LIN {X 0,Y 489.55,Z 664.789,A -85,B 0,C 180,E1 -6475.471,E2 -6475.471} C_VEL
LIN {X 0,Y 489.917,Z 653.885,A -85,B 0,C 180,E1 -6476.402,E2 -6476.402} C_VEL
LIN {X 0,Y 490.26,Z 643.208,A -85,B 0,C 180,E1 -6477.124,E2 -6477.124} C_VEL
LIN {X 0,Y 490.656,Z 630.33,A -85,B 0,C 180,E1 -6477.794,E2 -6477.794} C_VEL
LIN {X 0,Y 490.871,Z 617.995,A -85,B 0,C 180,E1 -6478.256,E2 -6478.256} C_VEL
LIN {X 0,Y 491.024,Z 605.317,A -85,B 0,C 180,E1 -6478.565,E2 -6478.565} C_VEL
LIN {X 0,Y 491.793,Z 513.634,A -85,B 0,C 180,E1 -6480,E2 -6480} C_VEL
LIN {X 0,Y 489.493,Z 503.257,A -85,B 0,C 180,E1 -6480.257,E2 -6480.257} C_VEL
LIN {X 0,Y 488.87,Z 498.779,A -85,B 0,C 180,E1 -6481.39,E2 -6481.39} C_VEL
LIN {X 0,Y 488.953,Z 498.58,A -85,B 0,C 180,E1 -6482.471,E2 -6482.471} C_VEL
LIN {X 0,Y 488.865,Z 498.591,A -85,B 0,C 180,E1 -6485.775,E2 -6485.775} C_VEL
LIN {X 0,Y 488.809,Z 498.595,A -85,B 0,C 180,E1 -6488.266,E2 -6488.266} C_VEL
LIN {X 0,Y 488.823,Z 498.596,A -85,B 0,C 180,E1 -6491.612,E2 -6491.612} C_VEL
LIN {X 0,Y 488.752,Z 498.606,A -85,B 0,C 180,E1 -6495.001,E2 -6495.001} C_VEL
LIN {X 0,Y 488.745,Z 498.601,A -85,B 0,C 180,E1 -6498.442,E2 -6498.442} C_VEL
LIN {X 0,Y 488.698,Z 498.614,A -85,B 0,C 180,E1 -6501.071,E2 -6501.071} C_VEL
LIN {X 0,Y 488.685,Z 498.61,A -85,B 0,C 180,E1 -6503.746,E2 -6503.746} C_VEL
LIN {X 0,Y 488.791,Z 498.6,A -85,B 0,C 180,E1 -6506.946,E2 -6506.946} C_VEL
LIN {X 0,Y 488.711,Z 498.603,A -85,B 0,C 180,E1 -6510.365,E2 -6510.365} C_VEL
LIN {X 0,Y 488.729,Z 498.604,A -85,B 0,C 180,E1 -6513.485,E2 -6513.485} C_VEL
LIN {X 0,Y 488.683,Z 498.607,A -85,B 0,C 180,E1 -6516.356,E2 -6516.356} C_VEL
LIN {X 0,Y 488.696,Z 498.612,A -85,B 0,C 180,E1 -6519.255,E2 -6519.255} C_VEL
LIN {X 0,Y 488.703,Z 498.607,A -85,B 0,C 180,E1 -6521.601,E2 -6521.601} C_VEL
LIN {X 0,Y 488.707,Z 498.612,A -85,B 0,C 180,E1 -6524.802,E2 -6524.802} C_VEL
LIN {X 0,Y 488.691,Z 498.612,A -85,B 0,C 180,E1 -6527.476,E2 -6527.476} C_VEL
LIN {X 0,Y 488.729,Z 498.605,A -85,B 0,C 180,E1 -6529.677,E2 -6529.677} C_VEL
LIN {X 0,Y 488.679,Z 498.616,A -85,B 0,C 180,E1 -6532.842,E2 -6532.842} C_VEL
LIN {X 0,Y 488.732,Z 498.605,A -85,B 0,C 180,E1 -6535.888,E2 -6535.888} C_VEL
LIN {X 0,Y 488.693,Z 498.618,A -85,B 0,C 180,E1 -6538.821,E2 -6538.821} C_VEL
LIN {X 0,Y 488.744,Z 498.606,A -85,B 0,C 180,E1 -6541.672,E2 -6541.672} C_VEL
LIN {X 0,Y 488.775,Z 498.713,A -85,B 0,C 180,E1 -6542.836,E2 -6542.836} C_VEL
LIN {X 0,Y 491.08,Z 510.544,A -85,B 0,C 180,E1 -6544.802,E2 -6544.802} C_VEL
LIN {X 0,Y 490.719,Z 523.768,A -85,B 0,C 180,E1 -6546.812,E2 -6546.812} C_VEL
LIN {X 0,Y 490.136,Z 541.34,A -85,B 0,C 180,E1 -6549.434,E2 -6549.434} C_VEL
LIN {X 0,Y 489.49,Z 563.398,A -85,B 0,C 180,E1 -6552.667,E2 -6552.667} C_VEL
LIN {X 0,Y 489.298,Z 570.739,A -85,B 0,C 180,E1 -6553.729,E2 -6553.729} C_VEL
LIN {X 0,Y 491.608,Z 589.498,A -85,B 0,C 180,E1 -6554.105,E2 -6554.105} C_VEL
LIN {X 0,Y 490.867,Z 681.432,A -85,B 0,C 180,E1 -6555.543,E2 -6555.543} C_VEL
LIN {X 0,Y 490.515,Z 695.071,A -85,B 0,C 180,E1 -6555.929,E2 -6555.929} C_VEL
LIN {X 0,Y 490.122,Z 707.959,A -85,B 0,C 180,E1 -6556.473,E2 -6556.473} C_VEL
LIN {X 0,Y 489.729,Z 720.461,A -85,B 0,C 180,E1 -6557.19,E2 -6557.19} C_VEL
LIN {X 0,Y 489.426,Z 731.262,A -85,B 0,C 180,E1 -6557.983,E2 -6557.983} C_VEL
LIN {X 0,Y 489.029,Z 741.567,A -85,B 0,C 180,E1 -6558.918,E2 -6558.918} C_VEL
LIN {X 0,Y 488.714,Z 750.11,A -85,B 0,C 180,E1 -6559.854,E2 -6559.854} C_VEL
LIN {X 0,Y 488.44,Z 757.894,A -85,B 0,C 180,E1 -6560.893,E2 -6560.893} C_VEL
LIN {X 0,Y 488.234,Z 765.619,A -85,B 0,C 180,E1 -6562.14,E2 -6562.14} C_VEL
LIN {X 0,Y 488.086,Z 772.223,A -85,B 0,C 180,E1 -6563.485,E2 -6563.485} C_VEL
LIN {X 0,Y 488.065,Z 776.673,A -85,B 0,C 180,E1 -6564.629,E2 -6564.629} C_VEL
LIN {X 0,Y 488.014,Z 780.377,A -85,B 0,C 180,E1 -6565.871,E2 -6565.871} C_VEL
LIN {X 0,Y 487.975,Z 782.291,A -85,B 0,C 180,E1 -6566.697,E2 -6566.697} C_VEL
LIN {X 0,Y 487.988,Z 783.763,A -85,B 0,C 180,E1 -6567.524,E2 -6567.524} C_VEL
LIN {X 0,Y 487.892,Z 784.813,A -85,B 0,C 180,E1 -6568.349,E2 -6568.349} C_VEL
LIN {X 0,Y 487.843,Z 785.455,A -85,B 0,C 180,E1 -6569.175,E2 -6569.175} C_VEL
LIN {X 0,Y 487.839,Z 785.68,A -85,B 0,C 180,E1 -6570,E2 -6570} C_VEL
LIN {X 0,Y 487.842,Z 785.48,A -85,B 0,C 180,E1 -6570.825,E2 -6570.825} C_VEL
LIN {X 0,Y 487.892,Z 784.879,A -85,B 0,C 180,E1 -6571.651,E2 -6571.651} C_VEL
LIN {X 0,Y 487.988,Z 783.864,A -85,B 0,C 180,E1 -6572.476,E2 -6572.476} C_VEL
LIN {X 0,Y 487.972,Z 782.417,A -85,B 0,C 180,E1 -6573.303,E2 -6573.303} C_VEL
LIN {X 0,Y 487.944,Z 779.439,A -85,B 0,C 180,E1 -6574.544,E2 -6574.544} C_VEL
LIN {X 0,Y 488.087,Z 775.402,A -85,B 0,C 180,E1 -6575.785,E2 -6575.785} C_VEL
LIN {X 0,Y 488.182,Z 769.169,A -85,B 0,C 180,E1 -6577.236,E2 -6577.236} C_VEL
LIN {X 0,Y 488.359,Z 762.353,A -85,B 0,C 180,E1 -6578.482,E2 -6578.482} C_VEL
LIN {X 0,Y 488.599,Z 753.841,A -85,B 0,C 180,E1 -6579.73,E2 -6579.73} C_VEL
LIN {X 0,Y 488.895,Z 745.105,A -85,B 0,C 180,E1 -6580.77,E2 -6580.77} C_VEL
LIN {X 0,Y 489.313,Z 735.631,A -85,B 0,C 180,E1 -6581.705,E2 -6581.705} C_VEL
LIN {X 0,Y 489.655,Z 724.66,A -85,B 0,C 180,E1 -6582.577,E2 -6582.577} C_VEL
LIN {X 0,Y 490.05,Z 713.845,A -85,B 0,C 180,E1 -6583.265,E2 -6583.265} C_VEL
LIN {X 0,Y 490.399,Z 702.302,A -85,B 0,C 180,E1 -6583.836,E2 -6583.836} C_VEL
LIN {X 0,Y 490.741,Z 690.007,A -85,B 0,C 180,E1 -6584.276,E2 -6584.276} C_VEL
LIN {X 0,Y 490.992,Z 676.488,A -85,B 0,C 180,E1 -6584.586,E2 -6584.586} C_VEL
LIN {X 0,Y 491.55,Z 587.504,A -85,B 0,C 180,E1 -6585.947,E2 -6585.947} C_VEL
LIN {X 0,Y 489.411,Z 571.971,A -85,B 0,C 180,E1 -6586.265,E2 -6586.265} C_VEL
LIN {X 0,Y 490.118,Z 548.737,A -85,B 0,C 180,E1 -6589.692,E2 -6589.692} C_VEL
LIN {X 0,Y 490.772,Z 529.767,A -85,B 0,C 180,E1 -6592.523,E2 -6592.523} C_VEL
LIN {X 0,Y 491.452,Z 513.716,A -85,B 0,C 180,E1 -6594.952,E2 -6594.952} C_VEL
LIN {X 0,Y 491.047,Z 509.509,A -85,B 0,C 180,E1 -6595.621,E2 -6595.621} C_VEL
LIN {X 0,Y 488.771,Z 498.604,A -85,B 0,C 180,E1 -6597.452,E2 -6597.452} C_VEL
LIN {X 0,Y 488.709,Z 498.608,A -85,B 0,C 180,E1 -6600.362,E2 -6600.362} C_VEL
LIN {X 0,Y 488.733,Z 498.607,A -85,B 0,C 180,E1 -6603.483,E2 -6603.483} C_VEL
LIN {X 0,Y 488.679,Z 498.607,A -85,B 0,C 180,E1 -6606.354,E2 -6606.354} C_VEL
LIN {X 0,Y 488.698,Z 498.602,A -85,B 0,C 180,E1 -6609.253,E2 -6609.253} C_VEL
LIN {X 0,Y 488.72,Z 498.607,A -85,B 0,C 180,E1 -6611.601,E2 -6611.601} C_VEL
LIN {X 0,Y 488.707,Z 498.606,A -85,B 0,C 180,E1 -6614.801,E2 -6614.801} C_VEL
LIN {X 0,Y 488.686,Z 498.608,A -85,B 0,C 180,E1 -6617.474,E2 -6617.474} C_VEL
LIN {X 0,Y 488.727,Z 498.605,A -85,B 0,C 180,E1 -6619.676,E2 -6619.676} C_VEL
LIN {X 0,Y 488.673,Z 498.608,A -85,B 0,C 180,E1 -6622.277,E2 -6622.277} C_VEL
LIN {X 0,Y 488.722,Z 498.607,A -85,B 0,C 180,E1 -6625.051,E2 -6625.051} C_VEL
LIN {X 0,Y 488.699,Z 498.603,A -85,B 0,C 180,E1 -6628.045,E2 -6628.045} C_VEL
LIN {X 0,Y 488.726,Z 498.601,A -85,B 0,C 180,E1 -6630.73,E2 -6630.73} C_VEL
LIN {X 0,Y 488.758,Z 498.6,A -85,B 0,C 180,E1 -6633.528,E2 -6633.528} C_VEL
LIN {X 0,Y 488.684,Z 498.598,A -85,B 0,C 180,E1 -6636.254,E2 -6636.254} C_VEL
LIN {X 0,Y 488.737,Z 498.609,A -85,B 0,C 180,E1 -6639.175,E2 -6639.175} C_VEL
LIN {X 0,Y 488.75,Z 498.597,A -85,B 0,C 180,E1 -6641.627,E2 -6641.627} C_VEL
LIN {X 0,Y 488.752,Z 498.598,A -85,B 0,C 180,E1 -6644.999,E2 -6644.999} C_VEL
LIN {X 0,Y 488.822,Z 498.591,A -85,B 0,C 180,E1 -6648.388,E2 -6648.388} C_VEL
LIN {X 0,Y 488.809,Z 498.584,A -85,B 0,C 180,E1 -6651.734,E2 -6651.734} C_VEL
LIN {X 0,Y 488.863,Z 498.584,A -85,B 0,C 180,E1 -6654.225,E2 -6654.225} C_VEL
LIN {X 0,Y 488.952,Z 498.574,A -85,B 0,C 180,E1 -6657.529,E2 -6657.529} C_VEL
LIN {X 0,Y 488.959,Z 498.561,A -85,B 0,C 180,E1 -6660,E2 -6660} C_VEL
LIN {X 0,Y 488.953,Z 498.572,A -85,B 0,C 180,E1 -6662.472,E2 -6662.472} C_VEL
LIN {X 0,Y 488.864,Z 498.584,A -85,B 0,C 180,E1 -6665.776,E2 -6665.776} C_VEL
LIN {X 0,Y 488.809,Z 498.583,A -85,B 0,C 180,E1 -6668.267,E2 -6668.267} C_VEL
LIN {X 0,Y 488.799,Z 498.595,A -85,B 0,C 180,E1 -6671.613,E2 -6671.613} C_VEL
LIN {X 0,Y 488.753,Z 498.6,A -85,B 0,C 180,E1 -6675.001,E2 -6675.001} C_VEL
LIN {X 0,Y 488.747,Z 498.599,A -85,B 0,C 180,E1 -6678.443,E2 -6678.443} C_VEL
LIN {X 0,Y 488.7,Z 498.611,A -85,B 0,C 180,E1 -6681.071,E2 -6681.071} C_VEL
LIN {X 0,Y 488.686,Z 498.603,A -85,B 0,C 180,E1 -6683.746,E2 -6683.746} C_VEL
LIN {X 0,Y 488.792,Z 498.602,A -85,B 0,C 180,E1 -6686.946,E2 -6686.946} C_VEL
LIN {X 0,Y 488.713,Z 498.601,A -85,B 0,C 180,E1 -6690.366,E2 -6690.366} C_VEL
LIN {X 0,Y 488.731,Z 498.603,A -85,B 0,C 180,E1 -6693.485,E2 -6693.485} C_VEL
LIN {X 0,Y 488.686,Z 498.608,A -85,B 0,C 180,E1 -6696.357,E2 -6696.357} C_VEL
LIN {X 0,Y 488.698,Z 498.61,A -85,B 0,C 180,E1 -6699.255,E2 -6699.255} C_VEL
LIN {X 0,Y 488.705,Z 498.609,A -85,B 0,C 180,E1 -6701.601,E2 -6701.601} C_VEL
LIN {X 0,Y 488.699,Z 498.606,A -85,B 0,C 180,E1 -6704.025,E2 -6704.025} C_VEL
LIN {X 0,Y 488.731,Z 498.608,A -85,B 0,C 180,E1 -6707.172,E2 -6707.172} C_VEL
LIN {X 0,Y 488.731,Z 498.603,A -85,B 0,C 180,E1 -6709.678,E2 -6709.678} C_VEL
LIN {X 0,Y 488.679,Z 498.615,A -85,B 0,C 180,E1 -6712.842,E2 -6712.842} C_VEL
LIN {X 0,Y 488.731,Z 498.603,A -85,B 0,C 180,E1 -6715.888,E2 -6715.888} C_VEL
LIN {X 0,Y 488.693,Z 498.611,A -85,B 0,C 180,E1 -6718.821,E2 -6718.821} C_VEL
LIN {X 0,Y 488.746,Z 498.603,A -85,B 0,C 180,E1 -6721.672,E2 -6721.672} C_VEL
LIN {X 0,Y 488.796,Z 498.602,A -85,B 0,C 180,E1 -6723.111,E2 -6723.111} C_VEL
LIN {X 0,Y 488.575,Z 499.275,A -85,B 0,C 180,E1 -6723.566,E2 -6723.566} C_VEL
LIN {X 0,Y 487.813,Z 501.458,A -85,B 0,C 180,E1 -6724.088,E2 -6724.088} C_VEL
LIN {X 0,Y 483.782,Z 512.802,A -85,B 0,C 180,E1 -6725.858,E2 -6725.858} C_VEL
LIN {X 0,Y 483.468,Z 515.113,A -85,B 0,C 180,E1 -6726.244,E2 -6726.244} C_VEL
LIN {X 0,Y 482.892,Z 533.439,A -85,B 0,C 180,E1 -6729.334,E2 -6729.334} C_VEL
LIN {X 0,Y 482.591,Z 546.967,A -85,B 0,C 180,E1 -6731.548,E2 -6731.548} C_VEL
LIN {X 0,Y 484.969,Z 561.064,A -85,B 0,C 180,E1 -6731.847,E2 -6731.847} C_VEL
LIN {X 0,Y 484.263,Z 656.005,A -85,B 0,C 180,E1 -6733.283,E2 -6733.283} C_VEL
LIN {X 0,Y 484.057,Z 669.122,A -85,B 0,C 180,E1 -6733.65,E2 -6733.65} C_VEL
LIN {X 0,Y 483.687,Z 681.903,A -85,B 0,C 180,E1 -6734.191,E2 -6734.191} C_VEL
LIN {X 0,Y 483.287,Z 693.124,A -85,B 0,C 180,E1 -6734.826,E2 -6734.826} C_VEL
LIN {X 0,Y 482.888,Z 703.46,A -85,B 0,C 180,E1 -6735.568,E2 -6735.568} C_VEL
LIN {X 0,Y 482.393,Z 714.084,A -85,B 0,C 180,E1 -6736.52,E2 -6736.52} C_VEL
LIN {X 0,Y 481.997,Z 724.342,A -85,B 0,C 180,E1 -6737.671,E2 -6737.671} C_VEL
LIN {X 0,Y 481.688,Z 732.834,A -85,B 0,C 180,E1 -6738.854,E2 -6738.854} C_VEL
LIN {X 0,Y 481.31,Z 740.173,A -85,B 0,C 180,E1 -6740.121,E2 -6740.121} C_VEL
LIN {X 0,Y 481.096,Z 746.945,A -85,B 0,C 180,E1 -6741.6,E2 -6741.6} C_VEL
LIN {X 0,Y 480.994,Z 751.387,A -85,B 0,C 180,E1 -6742.866,E2 -6742.866} C_VEL
LIN {X 0,Y 480.926,Z 754.743,A -85,B 0,C 180,E1 -6744.129,E2 -6744.129} C_VEL
LIN {X 0,Y 480.791,Z 757.67,A -85,B 0,C 180,E1 -6745.809,E2 -6745.809} C_VEL
LIN {X 0,Y 480.871,Z 758.544,A -85,B 0,C 180,E1 -6746.649,E2 -6746.649} C_VEL
LIN {X 0,Y 480.821,Z 759.001,A -85,B 0,C 180,E1 -6747.487,E2 -6747.487} C_VEL
LIN {X 0,Y 480.822,Z 759.052,A -85,B 0,C 180,E1 -6748.325,E2 -6748.325} C_VEL
LIN {X 0,Y 480.746,Z 758.024,A -85,B 0,C 180,E1 -6750,E2 -6750} C_VEL
LIN {X 0,Y 480.766,Z 756.885,A -85,B 0,C 180,E1 -6750.838,E2 -6750.838} C_VEL
LIN {X 0,Y 480.852,Z 755.339,A -85,B 0,C 180,E1 -6751.675,E2 -6751.675} C_VEL
LIN {X 0,Y 481.015,Z 752.226,A -85,B 0,C 180,E1 -6752.931,E2 -6752.931} C_VEL
LIN {X 0,Y 481.122,Z 748.071,A -85,B 0,C 180,E1 -6754.188,E2 -6754.188} C_VEL
LIN {X 0,Y 481.265,Z 741.773,A -85,B 0,C 180,E1 -6755.657,E2 -6755.657} C_VEL
LIN {X 0,Y 481.628,Z 735.259,A -85,B 0,C 180,E1 -6756.847,E2 -6756.847} C_VEL
LIN {X 0,Y 481.836,Z 727.805,A -85,B 0,C 180,E1 -6757.965,E2 -6757.965} C_VEL
LIN {X 0,Y 482.203,Z 719.295,A -85,B 0,C 180,E1 -6759.014,E2 -6759.014} C_VEL
LIN {X 0,Y 482.734,Z 708.869,A -85,B 0,C 180,E1 -6760.061,E2 -6760.061} C_VEL
LIN {X 0,Y 483.098,Z 698.445,A -85,B 0,C 180,E1 -6760.901,E2 -6760.901} C_VEL
LIN {X 0,Y 483.527,Z 686.901,A -85,B 0,C 180,E1 -6761.634,E2 -6761.634} C_VEL
LIN {X 0,Y 483.921,Z 675.067,A -85,B 0,C 180,E1 -6762.209,E2 -6762.209} C_VEL
LIN {X 0,Y 484.148,Z 662.145,A -85,B 0,C 180,E1 -6762.656,E2 -6762.656} C_VEL
LIN {X 0,Y 484.376,Z 648.3,A -85,B 0,C 180,E1 -6762.943,E2 -6762.943} C_VEL
LIN {X 0,Y 484.876,Z 560.303,A -85,B 0,C 180,E1 -6764.254,E2 -6764.254} C_VEL
LIN {X 0,Y 482.563,Z 546.856,A -85,B 0,C 180,E1 -6764.55,E2 -6764.55} C_VEL
LIN {X 0,Y 482.963,Z 529.781,A -85,B 0,C 180,E1 -6767.356,E2 -6767.356} C_VEL
LIN {X 0,Y 483.545,Z 510.287,A -85,B 0,C 180,E1 -6770.637,E2 -6770.637} C_VEL
LIN {X 0,Y 482.503,Z 503.71,A -85,B 0,C 180,E1 -6771.803,E2 -6771.803} C_VEL
LIN {X 0,Y 481.685,Z 499.49,A -85,B 0,C 180,E1 -6772.576,E2 -6772.576} C_VEL
LIN {X 0,Y 481.703,Z 499.481,A -85,B 0,C 180,E1 -6775.956,E2 -6775.956} C_VEL
LIN {X 0,Y 481.702,Z 499.485,A -85,B 0,C 180,E1 -6778.781,E2 -6778.781} C_VEL
LIN {X 0,Y 481.66,Z 499.486,A -85,B 0,C 180,E1 -6782.189,E2 -6782.189} C_VEL
LIN {X 0,Y 481.689,Z 499.483,A -85,B 0,C 180,E1 -6784.681,E2 -6784.681} C_VEL
LIN {X 0,Y 481.655,Z 499.484,A -85,B 0,C 180,E1 -6788.006,E2 -6788.006} C_VEL
LIN {X 0,Y 481.661,Z 499.488,A -85,B 0,C 180,E1 -6791.04,E2 -6791.04} C_VEL
LIN {X 0,Y 481.68,Z 499.483,A -85,B 0,C 180,E1 -6793.294,E2 -6793.294} C_VEL
LIN {X 0,Y 481.68,Z 499.485,A -85,B 0,C 180,E1 -6796.845,E2 -6796.845} C_VEL
LIN {X 0,Y 481.673,Z 499.483,A -85,B 0,C 180,E1 -6800.059,E2 -6800.059} C_VEL
LIN {X 0,Y 481.626,Z 499.491,A -85,B 0,C 180,E1 -6803.253,E2 -6803.253} C_VEL
LIN {X 0,Y 481.704,Z 499.484,A -85,B 0,C 180,E1 -6806.329,E2 -6806.329} C_VEL
LIN {X 0,Y 481.74,Z 499.495,A -85,B 0,C 180,E1 -6806.957,E2 -6806.957} C_VEL
LIN {X 0,Y 482.178,Z 502.037,A -85,B 0,C 180,E1 -6807.573,E2 -6807.573} C_VEL
LIN {X 0,Y 484.86,Z 513.987,A -85,B 0,C 180,E1 -6807.872,E2 -6807.872} C_VEL
LIN {X 0,Y 484.13,Z 608.315,A -85,B 0,C 180,E1 -6809.374,E2 -6809.374} C_VEL
LIN {X 0,Y 483.883,Z 621.472,A -85,B 0,C 180,E1 -6809.747,E2 -6809.747} C_VEL
LIN {X 0,Y 483.679,Z 633.972,A -85,B 0,C 180,E1 -6810.274,E2 -6810.274} C_VEL
LIN {X 0,Y 483.265,Z 646.179,A -85,B 0,C 180,E1 -6810.971,E2 -6810.971} C_VEL
LIN {X 0,Y 482.841,Z 657.038,A -85,B 0,C 180,E1 -6811.767,E2 -6811.767} C_VEL
LIN {X 0,Y 482.479,Z 667.159,A -85,B 0,C 180,E1 -6812.689,E2 -6812.689} C_VEL
LIN {X 0,Y 482.039,Z 677.233,A -85,B 0,C 180,E1 -6813.83,E2 -6813.83} C_VEL
LIN {X 0,Y 481.745,Z 685.374,A -85,B 0,C 180,E1 -6814.971,E2 -6814.971} C_VEL
LIN {X 0,Y 481.441,Z 693.216,A -85,B 0,C 180,E1 -6816.331,E2 -6816.331} C_VEL
LIN {X 0,Y 481.224,Z 699.311,A -85,B 0,C 180,E1 -6817.684,E2 -6817.684} C_VEL
LIN {X 0,Y 481.072,Z 704.569,A -85,B 0,C 180,E1 -6819.221,E2 -6819.221} C_VEL
LIN {X 0,Y 480.916,Z 707.444,A -85,B 0,C 180,E1 -6820.359,E2 -6820.359} C_VEL
LIN {X 0,Y 480.871,Z 709.94,A -85,B 0,C 180,E1 -6821.798,E2 -6821.798} C_VEL
LIN {X 0,Y 480.793,Z 711.099,A -85,B 0,C 180,E1 -6823.001,E2 -6823.001} C_VEL
LIN {X 0,Y 480.822,Z 711.43,A -85,B 0,C 180,E1 -6823.876,E2 -6823.876} C_VEL
LIN {X 0,Y 480.845,Z 711.334,A -85,B 0,C 180,E1 -6824.746,E2 -6824.746} C_VEL
LIN {X 0,Y 480.851,Z 710.776,A -85,B 0,C 180,E1 -6825.613,E2 -6825.613} C_VEL
LIN {X 0,Y 480.875,Z 709.814,A -85,B 0,C 180,E1 -6826.476,E2 -6826.476} C_VEL
LIN {X 0,Y 480.953,Z 708.435,A -85,B 0,C 180,E1 -6827.338,E2 -6827.338} C_VEL
LIN {X 0,Y 481.043,Z 705.478,A -85,B 0,C 180,E1 -6828.634,E2 -6828.634} C_VEL
LIN {X 0,Y 481.174,Z 701.505,A -85,B 0,C 180,E1 -6829.905,E2 -6829.905} C_VEL
LIN {X 0,Y 481.426,Z 695.323,A -85,B 0,C 180,E1 -6831.394,E2 -6831.394} C_VEL
LIN {X 0,Y 481.726,Z 687.998,A -85,B 0,C 180,E1 -6832.766,E2 -6832.766} C_VEL
LIN {X 0,Y 482.039,Z 680.194,A -85,B 0,C 180,E1 -6833.932,E2 -6833.932} C_VEL
LIN {X 0,Y 482.302,Z 671.585,A -85,B 0,C 180,E1 -6834.984,E2 -6834.984} C_VEL
LIN {X 0,Y 482.745,Z 660.949,A -85,B 0,C 180,E1 -6836.034,E2 -6836.034} C_VEL
LIN {X 0,Y 483.169,Z 650.341,A -85,B 0,C 180,E1 -6836.873,E2 -6836.873} C_VEL
LIN {X 0,Y 483.496,Z 640.424,A -85,B 0,C 180,E1 -6837.5,E2 -6837.5} C_VEL
LIN {X 0,Y 483.794,Z 627.481,A -85,B 0,C 180,E1 -6838.127,E2 -6838.127} C_VEL
LIN {X 0,Y 484.089,Z 614.439,A -85,B 0,C 180,E1 -6838.57,E2 -6838.57} C_VEL
LIN {X 0,Y 484.219,Z 601.944,A -85,B 0,C 180,E1 -6838.83,E2 -6838.83} C_VEL
LIN {X 0,Y 484.924,Z 514.261,A -85,B 0,C 180,E1 -6840.233,E2 -6840.233} C_VEL
LIN {X 0,Y 482.552,Z 503.84,A -85,B 0,C 180,E1 -6840.524,E2 -6840.524} C_VEL
LIN {X 0,Y 481.804,Z 499.472,A -85,B 0,C 180,E1 -6841.672,E2 -6841.672} C_VEL
LIN {X 0,Y 481.92,Z 499.456,A -85,B 0,C 180,E1 -6842.507,E2 -6842.507} C_VEL
LIN {X 0,Y 481.823,Z 499.468,A -85,B 0,C 180,E1 -6845.86,E2 -6845.86} C_VEL
LIN {X 0,Y 481.755,Z 499.474,A -85,B 0,C 180,E1 -6848.388,E2 -6848.388} C_VEL
LIN {X 0,Y 481.786,Z 499.471,A -85,B 0,C 180,E1 -6851.784,E2 -6851.784} C_VEL
LIN {X 0,Y 481.733,Z 499.481,A -85,B 0,C 180,E1 -6855.224,E2 -6855.224} C_VEL
LIN {X 0,Y 481.703,Z 499.48,A -85,B 0,C 180,E1 -6858.722,E2 -6858.722} C_VEL
LIN {X 0,Y 481.638,Z 499.491,A -85,B 0,C 180,E1 -6861.395,E2 -6861.395} C_VEL
LIN {X 0,Y 481.668,Z 499.482,A -85,B 0,C 180,E1 -6864.114,E2 -6864.114} C_VEL
LIN {X 0,Y 481.744,Z 499.478,A -85,B 0,C 180,E1 -6867.141,E2 -6867.141} C_VEL
LIN {X 0,Y 481.681,Z 499.48,A -85,B 0,C 180,E1 -6869.741,E2 -6869.741} C_VEL
LIN {X 0,Y 481.666,Z 499.483,A -85,B 0,C 180,E1 -6872.675,E2 -6872.675} C_VEL
LIN {X 0,Y 481.636,Z 499.485,A -85,B 0,C 180,E1 -6875.71,E2 -6875.71} C_VEL
LIN {X 0,Y 481.686,Z 499.485,A -85,B 0,C 180,E1 -6878.858,E2 -6878.858} C_VEL
LIN {X 0,Y 481.642,Z 499.486,A -85,B 0,C 180,E1 -6882.161,E2 -6882.161} C_VEL
LIN {X 0,Y 481.655,Z 499.487,A -85,B 0,C 180,E1 -6885.544,E2 -6885.544} C_VEL
LIN {X 0,Y 481.658,Z 499.486,A -85,B 0,C 180,E1 -6888.087,E2 -6888.087} C_VEL
LIN {X 0,Y 481.668,Z 499.488,A -85,B 0,C 180,E1 -6891.142,E2 -6891.142} C_VEL
LIN {X 0,Y 481.664,Z 499.491,A -85,B 0,C 180,E1 -6894.796,E2 -6894.796} C_VEL
LIN {X 0,Y 481.671,Z 499.49,A -85,B 0,C 180,E1 -6897.327,E2 -6897.327} C_VEL
LIN {X 0,Y 481.678,Z 499.488,A -85,B 0,C 180,E1 -6900.26,E2 -6900.26} C_VEL
LIN {X 0,Y 481.724,Z 499.583,A -85,B 0,C 180,E1 -6902.602,E2 -6902.602} C_VEL
LIN {X 0,Y 484.129,Z 511.692,A -85,B 0,C 180,E1 -6904.663,E2 -6904.663} C_VEL
LIN {X 0,Y 483.869,Z 522.387,A -85,B 0,C 180,E1 -6906.326,E2 -6906.326} C_VEL
LIN {X 0,Y 483.155,Z 542.273,A -85,B 0,C 180,E1 -6909.345,E2 -6909.345} C_VEL
LIN {X 0,Y 482.459,Z 564.242,A -85,B 0,C 180,E1 -6912.625,E2 -6912.625} C_VEL
LIN {X 0,Y 482.318,Z 569.981,A -85,B 0,C 180,E1 -6913.474,E2 -6913.474} C_VEL
LIN {X 0,Y 484.758,Z 589.981,A -85,B 0,C 180,E1 -6913.892,E2 -6913.892} C_VEL
LIN {X 0,Y 483.996,Z 680.253,A -85,B 0,C 180,E1 -6915.333,E2 -6915.333} C_VEL
LIN {X 0,Y 483.622,Z 693.277,A -85,B 0,C 180,E1 -6915.698,E2 -6915.698} C_VEL
LIN {X 0,Y 483.236,Z 705.973,A -85,B 0,C 180,E1 -6916.223,E2 -6916.223} C_VEL
LIN {X 0,Y 482.806,Z 717.844,A -85,B 0,C 180,E1 -6916.886,E2 -6916.886} C_VEL
LIN {X 0,Y 482.494,Z 729.198,A -85,B 0,C 180,E1 -6917.687,E2 -6917.687} C_VEL
LIN {X 0,Y 482.054,Z 740.067,A -85,B 0,C 180,E1 -6918.649,E2 -6918.649} C_VEL
LIN {X 0,Y 481.677,Z 749.678,A -85,B 0,C 180,E1 -6919.704,E2 -6919.704} C_VEL
LIN {X 0,Y 481.387,Z 757.526,A -85,B 0,C 180,E1 -6920.759,E2 -6920.759} C_VEL
LIN {X 0,Y 481.174,Z 765.167,A -85,B 0,C 180,E1 -6922.024,E2 -6922.024} C_VEL
LIN {X 0,Y 481.017,Z 771.283,A -85,B 0,C 180,E1 -6923.288,E2 -6923.288} C_VEL
LIN {X 0,Y 481.001,Z 776.127,A -85,B 0,C 180,E1 -6924.55,E2 -6924.55} C_VEL
LIN {X 0,Y 480.911,Z 779.792,A -85,B 0,C 180,E1 -6925.81,E2 -6925.81} C_VEL
LIN {X 0,Y 480.903,Z 781.715,A -85,B 0,C 180,E1 -6926.649,E2 -6926.649} C_VEL
LIN {X 0,Y 480.925,Z 783.201,A -85,B 0,C 180,E1 -6927.487,E2 -6927.487} C_VEL
LIN {X 0,Y 480.825,Z 784.256,A -85,B 0,C 180,E1 -6928.325,E2 -6928.325} C_VEL
LIN {X 0,Y 480.769,Z 784.905,A -85,B 0,C 180,E1 -6929.162,E2 -6929.162} C_VEL
LIN {X 0,Y 480.761,Z 785.14,A -85,B 0,C 180,E1 -6930,E2 -6930} C_VEL
LIN {X 0,Y 480.768,Z 784.944,A -85,B 0,C 180,E1 -6930.838,E2 -6930.838} C_VEL
LIN {X 0,Y 480.825,Z 784.339,A -85,B 0,C 180,E1 -6931.675,E2 -6931.675} C_VEL
LIN {X 0,Y 480.925,Z 783.322,A -85,B 0,C 180,E1 -6932.513,E2 -6932.513} C_VEL
LIN {X 0,Y 480.899,Z 781.872,A -85,B 0,C 180,E1 -6933.351,E2 -6933.351} C_VEL
LIN {X 0,Y 480.859,Z 778.887,A -85,B 0,C 180,E1 -6934.611,E2 -6934.611} C_VEL
LIN {X 0,Y 480.983,Z 774.845,A -85,B 0,C 180,E1 -6935.87,E2 -6935.87} C_VEL
LIN {X 0,Y 481.107,Z 768.598,A -85,B 0,C 180,E1 -6937.343,E2 -6937.343} C_VEL
LIN {X 0,Y 481.292,Z 761.756,A -85,B 0,C 180,E1 -6938.608,E2 -6938.608} C_VEL
LIN {X 0,Y 481.534,Z 753.224,A -85,B 0,C 180,E1 -6939.874,E2 -6939.874} C_VEL
LIN {X 0,Y 481.871,Z 744.459,A -85,B 0,C 180,E1 -6940.929,E2 -6940.929} C_VEL
LIN {X 0,Y 482.235,Z 735.012,A -85,B 0,C 180,E1 -6941.875,E2 -6941.875} C_VEL
LIN {X 0,Y 482.72,Z 723.355,A -85,B 0,C 180,E1 -6942.806,E2 -6942.806} C_VEL
LIN {X 0,Y 483.146,Z 711.178,A -85,B 0,C 180,E1 -6943.565,E2 -6943.565} C_VEL
LIN {X 0,Y 483.502,Z 698.859,A -85,B 0,C 180,E1 -6944.145,E2 -6944.145} C_VEL
LIN {X 0,Y 483.952,Z 685.369,A -85,B 0,C 180,E1 -6944.588,E2 -6944.588} C_VEL
LIN {X 0,Y 484.139,Z 670.223,A -85,B 0,C 180,E1 -6944.878,E2 -6944.878} C_VEL
LIN {X 0,Y 484.74,Z 588.484,A -85,B 0,C 180,E1 -6946.153,E2 -6946.153} C_VEL
LIN {X 0,Y 482.417,Z 571.336,A -85,B 0,C 180,E1 -6946.531,E2 -6946.531} C_VEL
LIN {X 0,Y 483.182,Z 548.255,A -85,B 0,C 180,E1 -6949.987,E2 -6949.987} C_VEL
LIN {X 0,Y 483.902,Z 529.32,A -85,B 0,C 180,E1 -6952.861,E2 -6952.861} C_VEL
LIN {X 0,Y 484.532,Z 514.74,A -85,B 0,C 180,E1 -6955.103,E2 -6955.103} C_VEL
LIN {X 0,Y 483.697,Z 508.822,A -85,B 0,C 180,E1 -6956.073,E2 -6956.073} C_VEL
LIN {X 0,Y 481.744,Z 499.48,A -85,B 0,C 180,E1 -6957.699,E2 -6957.699} C_VEL
LIN {X 0,Y 481.645,Z 499.49,A -85,B 0,C 180,E1 -6960.71,E2 -6960.71} C_VEL
LIN {X 0,Y 481.695,Z 499.482,A -85,B 0,C 180,E1 -6963.732,E2 -6963.732} C_VEL
LIN {X 0,Y 481.623,Z 499.489,A -85,B 0,C 180,E1 -6966.746,E2 -6966.746} C_VEL
LIN {X 0,Y 481.673,Z 499.48,A -85,B 0,C 180,E1 -6969.94,E2 -6969.94} C_VEL
LIN {X 0,Y 481.676,Z 499.484,A -85,B 0,C 180,E1 -6973.294,E2 -6973.294} C_VEL
LIN {X 0,Y 481.634,Z 499.49,A -85,B 0,C 180,E1 -6976.7,E2 -6976.7} C_VEL
LIN {X 0,Y 481.681,Z 499.481,A -85,B 0,C 180,E1 -6980.06,E2 -6980.06} C_VEL
LIN {X 0,Y 481.623,Z 499.488,A -85,B 0,C 180,E1 -6983.253,E2 -6983.253} C_VEL
LIN {X 0,Y 481.702,Z 499.478,A -85,B 0,C 180,E1 -6986.329,E2 -6986.329} C_VEL
LIN {X 0,Y 481.651,Z 499.483,A -85,B 0,C 180,E1 -6989.415,E2 -6989.415} C_VEL
LIN {X 0,Y 481.695,Z 499.478,A -85,B 0,C 180,E1 -6992.168,E2 -6992.168} C_VEL
LIN {X 0,Y 481.71,Z 499.478,A -85,B 0,C 180,E1 -6994.97,E2 -6994.97} C_VEL
LIN {X 0,Y 481.641,Z 499.485,A -85,B 0,C 180,E1 -6997.704,E2 -6997.704} C_VEL
LIN {X 0,Y 481.699,Z 499.478,A -85,B 0,C 180,E1 -7000.393,E2 -7000.393} C_VEL
LIN {X 0,Y 481.682,Z 499.477,A -85,B 0,C 180,E1 -7003.034,E2 -7003.034} C_VEL
LIN {X 0,Y 481.68,Z 499.481,A -85,B 0,C 180,E1 -7005.639,E2 -7005.639} C_VEL
LIN {X 0,Y 481.786,Z 499.467,A -85,B 0,C 180,E1 -7008.216,E2 -7008.216} C_VEL
LIN {X 0,Y 481.754,Z 499.463,A -85,B 0,C 180,E1 -7011.612,E2 -7011.612} C_VEL
LIN {X 0,Y 481.822,Z 499.461,A -85,B 0,C 180,E1 -7014.14,E2 -7014.14} C_VEL
LIN {X 0,Y 481.919,Z 499.45,A -85,B 0,C 180,E1 -7017.493,E2 -7017.493} C_VEL
LIN {X 0,Y 481.93,Z 499.436,A -85,B 0,C 180,E1 -7020,E2 -7020} C_VEL
LIN {X 0,Y 481.92,Z 499.449,A -85,B 0,C 180,E1 -7022.508,E2 -7022.508} C_VEL
LIN {X 0,Y 481.823,Z 499.461,A -85,B 0,C 180,E1 -7025.861,E2 -7025.861} C_VEL
LIN {X 0,Y 481.755,Z 499.461,A -85,B 0,C 180,E1 -7028.389,E2 -7028.389} C_VEL
LIN {X 0,Y 481.744,Z 499.473,A -85,B 0,C 180,E1 -7031.785,E2 -7031.785} C_VEL
LIN {X 0,Y 481.733,Z 499.47,A -85,B 0,C 180,E1 -7035.225,E2 -7035.225} C_VEL
LIN {X 0,Y 481.704,Z 499.479,A -85,B 0,C 180,E1 -7038.722,E2 -7038.722} C_VEL
LIN {X 0,Y 481.639,Z 499.486,A -85,B 0,C 180,E1 -7041.395,E2 -7041.395} C_VEL
LIN {X 0,Y 481.67,Z 499.476,A -85,B 0,C 180,E1 -7044.114,E2 -7044.114} C_VEL
LIN {X 0,Y 481.745,Z 499.478,A -85,B 0,C 180,E1 -7047.141,E2 -7047.141} C_VEL
LIN {X 0,Y 481.682,Z 499.476,A -85,B 0,C 180,E1 -7049.741,E2 -7049.741} C_VEL
LIN {X 0,Y 481.668,Z 499.486,A -85,B 0,C 180,E1 -7052.675,E2 -7052.675} C_VEL
LIN {X 0,Y 481.639,Z 499.486,A -85,B 0,C 180,E1 -7055.71,E2 -7055.71} C_VEL
LIN {X 0,Y 481.668,Z 499.489,A -85,B 0,C 180,E1 -7058.86,E2 -7058.86} C_VEL
LIN {X 0,Y 481.651,Z 499.487,A -85,B 0,C 180,E1 -7061.914,E2 -7061.914} C_VEL
LIN {X 0,Y 481.657,Z 499.485,A -85,B 0,C 180,E1 -7064.458,E2 -7064.458} C_VEL
LIN {X 0,Y 481.682,Z 499.486,A -85,B 0,C 180,E1 -7066.847,E2 -7066.847} C_VEL
LIN {X 0,Y 481.676,Z 499.481,A -85,B 0,C 180,E1 -7070.061,E2 -7070.061} C_VEL
LIN {X 0,Y 481.625,Z 499.493,A -85,B 0,C 180,E1 -7073.254,E2 -7073.254} C_VEL
LIN {X 0,Y 481.71,Z 499.479,A -85,B 0,C 180,E1 -7076.331,E2 -7076.331} C_VEL
LIN {X 0,Y 481.652,Z 499.488,A -85,B 0,C 180,E1 -7079.418,E2 -7079.418} C_VEL
LIN {X 0,Y 481.702,Z 499.48,A -85,B 0,C 180,E1 -7082.169,E2 -7082.169} C_VEL
LIN {X 0,Y 481.787,Z 499.513,A -85,B 0,C 180,E1 -7083.495,E2 -7083.495} C_VEL
LIN {X 0,Y 483.515,Z 509.606,A -85,B 0,C 180,E1 -7085.299,E2 -7085.299} C_VEL
LIN {X 0,Y 483.468,Z 515.113,A -85,B 0,C 180,E1 -7086.244,E2 -7086.244} C_VEL
LIN {X 0,Y 482.692,Z 518.578,A -85,B 0,C 180,E1 -7086.804,E2 -7086.804} C_VEL
LIN {X 0,Y 476.721,Z 530.43,A -85,B 0,C 180,E1 -7088.57,E2 -7088.57} C_VEL
LIN {X 0,Y 475.961,Z 533.953,A -85,B 0,C 180,E1 -7089.137,E2 -7089.137} C_VEL
LIN {X 0,Y 475.667,Z 546.954,A -85,B 0,C 180,E1 -7091.283,E2 -7091.283} C_VEL
LIN {X 0,Y 478.167,Z 561.911,A -85,B 0,C 180,E1 -7091.616,E2 -7091.616} C_VEL
LIN {X 0,Y 477.415,Z 655.957,A -85,B 0,C 180,E1 -7093.06,E2 -7093.06} C_VEL
LIN {X 0,Y 477.185,Z 668.456,A -85,B 0,C 180,E1 -7093.407,E2 -7093.407} C_VEL
LIN {X 0,Y 476.879,Z 680.479,A -85,B 0,C 180,E1 -7093.904,E2 -7093.904} C_VEL
LIN {X 0,Y 476.397,Z 692.874,A -85,B 0,C 180,E1 -7094.601,E2 -7094.601} C_VEL
LIN {X 0,Y 475.908,Z 704.623,A -85,B 0,C 180,E1 -7095.461,E2 -7095.461} C_VEL
LIN {X 0,Y 475.397,Z 715.032,A -85,B 0,C 180,E1 -7096.427,E2 -7096.427} C_VEL
LIN {X 0,Y 474.995,Z 724.928,A -85,B 0,C 180,E1 -7097.565,E2 -7097.565} C_VEL
LIN {X 0,Y 474.674,Z 732.841,A -85,B 0,C 180,E1 -7098.687,E2 -7098.687} C_VEL
LIN {X 0,Y 474.262,Z 740.211,A -85,B 0,C 180,E1 -7099.973,E2 -7099.973} C_VEL
LIN {X 0,Y 474.034,Z 747.016,A -85,B 0,C 180,E1 -7101.474,E2 -7101.474} C_VEL
LIN {X 0,Y 473.919,Z 751.488,A -85,B 0,C 180,E1 -7102.759,E2 -7102.759} C_VEL
LIN {X 0,Y 473.839,Z 754.868,A -85,B 0,C 180,E1 -7104.041,E2 -7104.041} C_VEL
LIN {X 0,Y 473.776,Z 756.548,A -85,B 0,C 180,E1 -7104.894,E2 -7104.894} C_VEL
LIN {X 0,Y 473.777,Z 758.708,A -85,B 0,C 180,E1 -7106.598,E2 -7106.598} C_VEL
LIN {X 0,Y 473.739,Z 759.186,A -85,B 0,C 180,E1 -7107.449,E2 -7107.449} C_VEL
LIN {X 0,Y 473.689,Z 758.934,A -85,B 0,C 180,E1 -7109.15,E2 -7109.15} C_VEL
LIN {X 0,Y 473.672,Z 758.243,A -85,B 0,C 180,E1 -7110,E2 -7110} C_VEL
LIN {X 0,Y 473.695,Z 757.123,A -85,B 0,C 180,E1 -7110.85,E2 -7110.85} C_VEL
LIN {X 0,Y 473.786,Z 755.588,A -85,B 0,C 180,E1 -7111.7,E2 -7111.7} C_VEL
LIN {X 0,Y 473.953,Z 752.497,A -85,B 0,C 180,E1 -7112.975,E2 -7112.975} C_VEL
LIN {X 0,Y 474.067,Z 748.365,A -85,B 0,C 180,E1 -7114.251,E2 -7114.251} C_VEL
LIN {X 0,Y 474.197,Z 742.098,A -85,B 0,C 180,E1 -7115.741,E2 -7115.741} C_VEL
LIN {X 0,Y 474.597,Z 735.411,A -85,B 0,C 180,E1 -7116.983,E2 -7116.983} C_VEL
LIN {X 0,Y 474.891,Z 726.622,A -85,B 0,C 180,E1 -7118.296,E2 -7118.296} C_VEL
LIN {X 0,Y 475.317,Z 717.838,A -85,B 0,C 180,E1 -7119.36,E2 -7119.36} C_VEL
LIN {X 0,Y 475.819,Z 708.151,A -85,B 0,C 180,E1 -7120.317,E2 -7120.317} C_VEL
LIN {X 0,Y 476.238,Z 697.481,A -85,B 0,C 180,E1 -7121.168,E2 -7121.168} C_VEL
LIN {X 0,Y 476.634,Z 685.65,A -85,B 0,C 180,E1 -7121.913,E2 -7121.913} C_VEL
LIN {X 0,Y 477.098,Z 673.223,A -85,B 0,C 180,E1 -7122.495,E2 -7122.495} C_VEL
LIN {X 0,Y 477.324,Z 660.21,A -85,B 0,C 180,E1 -7122.921,E2 -7122.921} C_VEL
LIN {X 0,Y 477.534,Z 646.459,A -85,B 0,C 180,E1 -7123.186,E2 -7123.186} C_VEL
LIN {X 0,Y 478.076,Z 561.297,A -85,B 0,C 180,E1 -7124.472,E2 -7124.472} C_VEL
LIN {X 0,Y 475.603,Z 546.948,A -85,B 0,C 180,E1 -7124.795,E2 -7124.795} C_VEL
LIN {X 0,Y 475.995,Z 531.171,A -85,B 0,C 180,E1 -7127.396,E2 -7127.396} C_VEL
LIN {X 0,Y 476.615,Z 511.543,A -85,B 0,C 180,E1 -7130.725,E2 -7130.725} C_VEL
LIN {X 0,Y 475.011,Z 502.231,A -85,B 0,C 180,E1 -7132.394,E2 -7132.394} C_VEL
LIN {X 0,Y 474.651,Z 500.368,A -85,B 0,C 180,E1 -7132.743,E2 -7132.743} C_VEL
LIN {X 0,Y 474.673,Z 500.361,A -85,B 0,C 180,E1 -7135.427,E2 -7135.427} C_VEL
LIN {X 0,Y 474.648,Z 500.359,A -85,B 0,C 180,E1 -7138.282,E2 -7138.282} C_VEL
LIN {X 0,Y 474.602,Z 500.369,A -85,B 0,C 180,E1 -7141.217,E2 -7141.217} C_VEL
LIN {X 0,Y 474.632,Z 500.359,A -85,B 0,C 180,E1 -7144.24,E2 -7144.24} C_VEL
LIN {X 0,Y 474.59,Z 500.367,A -85,B 0,C 180,E1 -7147.383,E2 -7147.383} C_VEL
LIN {X 0,Y 474.627,Z 500.358,A -85,B 0,C 180,E1 -7149.647,E2 -7149.647} C_VEL
LIN {X 0,Y 474.646,Z 500.364,A -85,B 0,C 180,E1 -7152.929,E2 -7152.929} C_VEL
LIN {X 0,Y 474.615,Z 500.356,A -85,B 0,C 180,E1 -7155.895,E2 -7155.895} C_VEL
LIN {X 0,Y 474.629,Z 500.365,A -85,B 0,C 180,E1 -7159.039,E2 -7159.039} C_VEL
LIN {X 0,Y 474.607,Z 500.363,A -85,B 0,C 180,E1 -7161.703,E2 -7161.703} C_VEL
LIN {X 0,Y 474.626,Z 500.367,A -85,B 0,C 180,E1 -7164.725,E2 -7164.725} C_VEL
LIN {X 0,Y 474.721,Z 500.451,A -85,B 0,C 180,E1 -7166.832,E2 -7166.832} C_VEL
LIN {X 0,Y 475.094,Z 502.632,A -85,B 0,C 180,E1 -7167.338,E2 -7167.338} C_VEL
LIN {X 0,Y 477.852,Z 513.777,A -85,B 0,C 180,E1 -7167.622,E2 -7167.622} C_VEL
LIN {X 0,Y 478.137,Z 517.504,A -85,B 0,C 180,E1 -7167.694,E2 -7167.694} C_VEL
LIN {X 0,Y 477.244,Z 609.282,A -85,B 0,C 180,E1 -7169.189,E2 -7169.189} C_VEL
LIN {X 0,Y 476.964,Z 623.116,A -85,B 0,C 180,E1 -7169.598,E2 -7169.598} C_VEL
LIN {X 0,Y 476.759,Z 634.781,A -85,B 0,C 180,E1 -7170.107,E2 -7170.107} C_VEL
LIN {X 0,Y 476.361,Z 645.79,A -85,B 0,C 180,E1 -7170.739,E2 -7170.739} C_VEL
LIN {X 0,Y 475.912,Z 656.968,A -85,B 0,C 180,E1 -7171.559,E2 -7171.559} C_VEL
LIN {X 0,Y 475.502,Z 667.864,A -85,B 0,C 180,E1 -7172.561,E2 -7172.561} C_VEL
LIN {X 0,Y 475.078,Z 677.407,A -85,B 0,C 180,E1 -7173.653,E2 -7173.653} C_VEL
LIN {X 0,Y 474.742,Z 685.615,A -85,B 0,C 180,E1 -7174.81,E2 -7174.81} C_VEL
LIN {X 0,Y 474.413,Z 693.522,A -85,B 0,C 180,E1 -7176.191,E2 -7176.191} C_VEL
LIN {X 0,Y 474.227,Z 698.761,A -85,B 0,C 180,E1 -7177.336,E2 -7177.336} C_VEL
LIN {X 0,Y 474.062,Z 703.744,A -85,B 0,C 180,E1 -7178.702,E2 -7178.702} C_VEL
LIN {X 0,Y 473.896,Z 707.428,A -85,B 0,C 180,E1 -7180.056,E2 -7180.056} C_VEL
LIN {X 0,Y 473.796,Z 710.353,A -85,B 0,C 180,E1 -7181.679,E2 -7181.679} C_VEL
LIN {X 0,Y 473.722,Z 711.491,A -85,B 0,C 180,E1 -7182.739,E2 -7182.739} C_VEL
LIN {X 0,Y 473.744,Z 711.919,A -85,B 0,C 180,E1 -7183.628,E2 -7183.628} C_VEL
LIN {X 0,Y 473.766,Z 711.92,A -85,B 0,C 180,E1 -7184.624,E2 -7184.624} C_VEL
LIN {X 0,Y 473.785,Z 711.54,A -85,B 0,C 180,E1 -7185.394,E2 -7185.394} C_VEL
LIN {X 0,Y 473.787,Z 710.678,A -85,B 0,C 180,E1 -7186.27,E2 -7186.27} C_VEL
LIN {X 0,Y 473.857,Z 709.396,A -85,B 0,C 180,E1 -7187.145,E2 -7187.145} C_VEL
LIN {X 0,Y 473.944,Z 707.403,A -85,B 0,C 180,E1 -7188.146,E2 -7188.146} C_VEL
LIN {X 0,Y 474.099,Z 702.852,A -85,B 0,C 180,E1 -7189.753,E2 -7189.753} C_VEL
LIN {X 0,Y 474.306,Z 697.908,A -85,B 0,C 180,E1 -7191.049,E2 -7191.049} C_VEL
LIN {X 0,Y 474.544,Z 691.685,A -85,B 0,C 180,E1 -7192.34,E2 -7192.34} C_VEL
LIN {X 0,Y 474.918,Z 683.858,A -85,B 0,C 180,E1 -7193.628,E2 -7193.628} C_VEL
LIN {X 0,Y 475.195,Z 675.908,A -85,B 0,C 180,E1 -7194.696,E2 -7194.696} C_VEL
LIN {X 0,Y 475.666,Z 666.161,A -85,B 0,C 180,E1 -7195.763,E2 -7195.763} C_VEL
LIN {X 0,Y 475.981,Z 656.661,A -85,B 0,C 180,E1 -7196.614,E2 -7196.614} C_VEL
LIN {X 0,Y 476.378,Z 646.41,A -85,B 0,C 180,E1 -7197.357,E2 -7197.357} C_VEL
LIN {X 0,Y 476.797,Z 634.13,A -85,B 0,C 180,E1 -7198.046,E2 -7198.046} C_VEL
LIN {X 0,Y 477.08,Z 621.341,A -85,B 0,C 180,E1 -7198.575,E2 -7198.575} C_VEL
LIN {X 0,Y 477.279,Z 608.972,A -85,B 0,C 180,E1 -7198.919,E2 -7198.919} C_VEL
LIN {X 0,Y 478.194,Z 515.267,A -85,B 0,C 180,E1 -7200.469,E2 -7200.469} C_VEL
LIN {X 0,Y 475.57,Z 504.572,A -85,B 0,C 180,E1 -7200.767,E2 -7200.767} C_VEL
LIN {X 0,Y 474.803,Z 500.345,A -85,B 0,C 180,E1 -7201.908,E2 -7201.908} C_VEL
LIN {X 0,Y 474.679,Z 500.36,A -85,B 0,C 180,E1 -7203.395,E2 -7203.395} C_VEL
LIN {X 0,Y 474.783,Z 500.344,A -85,B 0,C 180,E1 -7205.947,E2 -7205.947} C_VEL
LIN {X 0,Y 474.72,Z 500.351,A -85,B 0,C 180,E1 -7208.514,E2 -7208.514} C_VEL
LIN {X 0,Y 474.729,Z 500.349,A -85,B 0,C 180,E1 -7211.962,E2 -7211.962} C_VEL
LIN {X 0,Y 474.671,Z 500.357,A -85,B 0,C 180,E1 -7215.768,E2 -7215.768} C_VEL
LIN {X 0,Y 474.656,Z 500.361,A -85,B 0,C 180,E1 -7219.011,E2 -7219.011} C_VEL
LIN {X 0,Y 474.581,Z 500.367,A -85,B 0,C 180,E1 -7221.729,E2 -7221.729} C_VEL
LIN {X 0,Y 474.65,Z 500.358,A -85,B 0,C 180,E1 -7224.493,E2 -7224.493} C_VEL
LIN {X 0,Y 474.691,Z 500.354,A -85,B 0,C 180,E1 -7227.339,E2 -7227.339} C_VEL
LIN {X 0,Y 474.603,Z 500.365,A -85,B 0,C 180,E1 -7230.812,E2 -7230.812} C_VEL
LIN {X 0,Y 474.631,Z 500.357,A -85,B 0,C 180,E1 -7233.985,E2 -7233.985} C_VEL
LIN {X 0,Y 474.569,Z 500.371,A -85,B 0,C 180,E1 -7236.901,E2 -7236.901} C_VEL
LIN {X 0,Y 474.622,Z 500.361,A -85,B 0,C 180,E1 -7239.648,E2 -7239.648} C_VEL
LIN {X 0,Y 474.61,Z 500.369,A -85,B 0,C 180,E1 -7242.935,E2 -7242.935} C_VEL
LIN {X 0,Y 474.61,Z 500.363,A -85,B 0,C 180,E1 -7245.897,E2 -7245.897} C_VEL
LIN {X 0,Y 474.629,Z 500.367,A -85,B 0,C 180,E1 -7249.041,E2 -7249.041} C_VEL
LIN {X 0,Y 474.608,Z 500.364,A -85,B 0,C 180,E1 -7251.705,E2 -7251.705} C_VEL
LIN {X 0,Y 474.626,Z 500.367,A -85,B 0,C 180,E1 -7254.727,E2 -7254.727} C_VEL
LIN {X 0,Y 474.636,Z 500.364,A -85,B 0,C 180,E1 -7257.789,E2 -7257.789} C_VEL
LIN {X 0,Y 474.623,Z 500.368,A -85,B 0,C 180,E1 -7260.885,E2 -7260.885} C_VEL
LIN {X 0,Y 474.69,Z 500.494,A -85,B 0,C 180,E1 -7262.367,E2 -7262.367} C_VEL
LIN {X 0,Y 477.074,Z 512.147,A -85,B 0,C 180,E1 -7264.401,E2 -7264.401} C_VEL
LIN {X 0,Y 477.266,Z 516.986,A -85,B 0,C 180,E1 -7265.186,E2 -7265.186} C_VEL
LIN {X 0,Y 476.353,Z 538.811,A -85,B 0,C 180,E1 -7268.583,E2 -7268.583} C_VEL
LIN {X 0,Y 475.541,Z 560.748,A -85,B 0,C 180,E1 -7271.92,E2 -7271.92} C_VEL
LIN {X 0,Y 475.32,Z 569.485,A -85,B 0,C 180,E1 -7273.225,E2 -7273.225} C_VEL
LIN {X 0,Y 477.913,Z 591.056,A -85,B 0,C 180,E1 -7273.685,E2 -7273.685} C_VEL
LIN {X 0,Y 477.096,Z 680.236,A -85,B 0,C 180,E1 -7275.143,E2 -7275.143} C_VEL
LIN {X 0,Y 476.686,Z 693.807,A -85,B 0,C 180,E1 -7275.54,E2 -7275.54} C_VEL
LIN {X 0,Y 476.18,Z 708.461,A -85,B 0,C 180,E1 -7276.178,E2 -7276.178} C_VEL
LIN {X 0,Y 475.772,Z 720.389,A -85,B 0,C 180,E1 -7276.873,E2 -7276.873} C_VEL
LIN {X 0,Y 475.426,Z 731.449,A -85,B 0,C 180,E1 -7277.704,E2 -7277.704} C_VEL
LIN {X 0,Y 474.98,Z 742.006,A -85,B 0,C 180,E1 -7278.694,E2 -7278.694} C_VEL
LIN {X 0,Y 474.56,Z 751.168,A -85,B 0,C 180,E1 -7279.764,E2 -7279.764} C_VEL
LIN {X 0,Y 474.24,Z 760.074,A -85,B 0,C 180,E1 -7281.048,E2 -7281.048} C_VEL
LIN {X 0,Y 474.035,Z 767.195,A -85,B 0,C 180,E1 -7282.332,E2 -7282.332} C_VEL
LIN {X 0,Y 473.895,Z 772.528,A -85,B 0,C 180,E1 -7283.53,E2 -7283.53} C_VEL
LIN {X 0,Y 473.847,Z 777.277,A -85,B 0,C 180,E1 -7284.895,E2 -7284.895} C_VEL
LIN {X 0,Y 473.804,Z 779.608,A -85,B 0,C 180,E1 -7285.747,E2 -7285.747} C_VEL
LIN {X 0,Y 473.814,Z 781.507,A -85,B 0,C 180,E1 -7286.599,E2 -7286.599} C_VEL
LIN {X 0,Y 473.834,Z 782.941,A -85,B 0,C 180,E1 -7287.45,E2 -7287.45} C_VEL
LIN {X 0,Y 473.76,Z 783.949,A -85,B 0,C 180,E1 -7288.3,E2 -7288.3} C_VEL
LIN {X 0,Y 473.687,Z 784.785,A -85,B 0,C 180,E1 -7290,E2 -7290} C_VEL
LIN {X 0,Y 473.76,Z 783.946,A -85,B 0,C 180,E1 -7291.7,E2 -7291.7} C_VEL
LIN {X 0,Y 473.834,Z 782.937,A -85,B 0,C 180,E1 -7292.55,E2 -7292.55} C_VEL
LIN {X 0,Y 473.827,Z 781.502,A -85,B 0,C 180,E1 -7293.401,E2 -7293.401} C_VEL
LIN {X 0,Y 473.78,Z 778.514,A -85,B 0,C 180,E1 -7294.68,E2 -7294.68} C_VEL
LIN {X 0,Y 473.883,Z 774.46,A -85,B 0,C 180,E1 -7295.959,E2 -7295.959} C_VEL
LIN {X 0,Y 474.016,Z 768.203,A -85,B 0,C 180,E1 -7297.454,E2 -7297.454} C_VEL
LIN {X 0,Y 474.216,Z 761.357,A -85,B 0,C 180,E1 -7298.737,E2 -7298.737} C_VEL
LIN {X 0,Y 474.441,Z 754.367,A -85,B 0,C 180,E1 -7299.808,E2 -7299.808} C_VEL
LIN {X 0,Y 474.79,Z 745.916,A -85,B 0,C 180,E1 -7300.878,E2 -7300.878} C_VEL
LIN {X 0,Y 475.188,Z 735.42,A -85,B 0,C 180,E1 -7301.95,E2 -7301.95} C_VEL
LIN {X 0,Y 475.635,Z 725.239,A -85,B 0,C 180,E1 -7302.805,E2 -7302.805} C_VEL
LIN {X 0,Y 476.077,Z 714.131,A -85,B 0,C 180,E1 -7303.553,E2 -7303.553} C_VEL
LIN {X 0,Y 476.521,Z 701.836,A -85,B 0,C 180,E1 -7304.193,E2 -7304.193} C_VEL
LIN {X 0,Y 476.897,Z 688.937,A -85,B 0,C 180,E1 -7304.672,E2 -7304.672} C_VEL
LIN {X 0,Y 477.221,Z 675.422,A -85,B 0,C 180,E1 -7304.989,E2 -7304.989} C_VEL
LIN {X 0,Y 477.811,Z 588.468,A -85,B 0,C 180,E1 -7306.385,E2 -7306.385} C_VEL
LIN {X 0,Y 475.425,Z 570.845,A -85,B 0,C 180,E1 -7306.781,E2 -7306.781} C_VEL
LIN {X 0,Y 476.202,Z 549.234,A -85,B 0,C 180,E1 -7310.067,E2 -7310.067} C_VEL
LIN {X 0,Y 476.951,Z 530.326,A -85,B 0,C 180,E1 -7312.984,E2 -7312.984} C_VEL
LIN {X 0,Y 477.623,Z 515.726,A -85,B 0,C 180,E1 -7315.259,E2 -7315.259} C_VEL
LIN {X 0,Y 476.65,Z 509.777,A -85,B 0,C 180,E1 -7316.252,E2 -7316.252} C_VEL
LIN {X 0,Y 474.692,Z 500.357,A -85,B 0,C 180,E1 -7317.896,E2 -7317.896} C_VEL
LIN {X 0,Y 474.598,Z 500.371,A -85,B 0,C 180,E1 -7321.217,E2 -7321.217} C_VEL
LIN {X 0,Y 474.629,Z 500.36,A -85,B 0,C 180,E1 -7324.24,E2 -7324.24} C_VEL
LIN {X 0,Y 474.587,Z 500.354,A -85,B 0,C 180,E1 -7327.383,E2 -7327.383} C_VEL
LIN {X 0,Y 474.625,Z 500.36,A -85,B 0,C 180,E1 -7329.647,E2 -7329.647} C_VEL
LIN {X 0,Y 474.64,Z 500.363,A -85,B 0,C 180,E1 -7332.93,E2 -7332.93} C_VEL
LIN {X 0,Y 474.604,Z 500.364,A -85,B 0,C 180,E1 -7335.894,E2 -7335.894} C_VEL
LIN {X 0,Y 474.635,Z 500.359,A -85,B 0,C 180,E1 -7339.038,E2 -7339.038} C_VEL
LIN {X 0,Y 474.609,Z 500.362,A -85,B 0,C 180,E1 -7341.703,E2 -7341.703} C_VEL
LIN {X 0,Y 474.624,Z 500.359,A -85,B 0,C 180,E1 -7344.726,E2 -7344.726} C_VEL
LIN {X 0,Y 474.63,Z 500.356,A -85,B 0,C 180,E1 -7347.787,E2 -7347.787} C_VEL
LIN {X 0,Y 474.624,Z 500.359,A -85,B 0,C 180,E1 -7350.882,E2 -7350.882} C_VEL
LIN {X 0,Y 474.658,Z 500.355,A -85,B 0,C 180,E1 -7353.628,E2 -7353.628} C_VEL
LIN {X 0,Y 474.627,Z 500.351,A -85,B 0,C 180,E1 -7356.641,E2 -7356.641} C_VEL
LIN {X 0,Y 474.648,Z 500.356,A -85,B 0,C 180,E1 -7360.089,E2 -7360.089} C_VEL
LIN {X 0,Y 474.642,Z 500.355,A -85,B 0,C 180,E1 -7362.774,E2 -7362.774} C_VEL
LIN {X 0,Y 474.639,Z 500.361,A -85,B 0,C 180,E1 -7365.421,E2 -7365.421} C_VEL
LIN {X 0,Y 474.73,Z 500.346,A -85,B 0,C 180,E1 -7368.038,E2 -7368.038} C_VEL
LIN {X 0,Y 474.72,Z 500.34,A -85,B 0,C 180,E1 -7371.486,E2 -7371.486} C_VEL
LIN {X 0,Y 474.782,Z 500.337,A -85,B 0,C 180,E1 -7374.053,E2 -7374.053} C_VEL
LIN {X 0,Y 474.886,Z 500.327,A -85,B 0,C 180,E1 -7377.456,E2 -7377.456} C_VEL
LIN {X 0,Y 474.868,Z 500.32,A -85,B 0,C 180,E1 -7380.848,E2 -7380.848} C_VEL
LIN {X 0,Y 474.887,Z 500.325,A -85,B 0,C 180,E1 -7382.545,E2 -7382.545} C_VEL
LIN {X 0,Y 474.783,Z 500.337,A -85,B 0,C 180,E1 -7385.948,E2 -7385.948} C_VEL
LIN {X 0,Y 474.72,Z 500.338,A -85,B 0,C 180,E1 -7388.514,E2 -7388.514} C_VEL
LIN {X 0,Y 474.696,Z 500.351,A -85,B 0,C 180,E1 -7391.963,E2 -7391.963} C_VEL
LIN {X 0,Y 474.691,Z 500.344,A -85,B 0,C 180,E1 -7395.456,E2 -7395.456} C_VEL
LIN {X 0,Y 474.658,Z 500.361,A -85,B 0,C 180,E1 -7399.011,E2 -7399.011} C_VEL
LIN {X 0,Y 474.582,Z 500.362,A -85,B 0,C 180,E1 -7401.73,E2 -7401.73} C_VEL
LIN {X 0,Y 474.652,Z 500.352,A -85,B 0,C 180,E1 -7404.494,E2 -7404.494} C_VEL
LIN {X 0,Y 474.692,Z 500.354,A -85,B 0,C 180,E1 -7407.34,E2 -7407.34} C_VEL
LIN {X 0,Y 474.611,Z 500.361,A -85,B 0,C 180,E1 -7410.814,E2 -7410.814} C_VEL
LIN {X 0,Y 474.633,Z 500.356,A -85,B 0,C 180,E1 -7413.985,E2 -7413.985} C_VEL
LIN {X 0,Y 474.573,Z 500.372,A -85,B 0,C 180,E1 -7416.901,E2 -7416.901} C_VEL
LIN {X 0,Y 474.624,Z 500.36,A -85,B 0,C 180,E1 -7419.649,E2 -7419.649} C_VEL
LIN {X 0,Y 474.636,Z 500.365,A -85,B 0,C 180,E1 -7422.932,E2 -7422.932} C_VEL
LIN {X 0,Y 474.616,Z 500.362,A -85,B 0,C 180,E1 -7425.897,E2 -7425.897} C_VEL
LIN {X 0,Y 474.631,Z 500.364,A -85,B 0,C 180,E1 -7429.041,E2 -7429.041} C_VEL
LIN {X 0,Y 474.61,Z 500.361,A -85,B 0,C 180,E1 -7431.705,E2 -7431.705} C_VEL
LIN {X 0,Y 474.624,Z 500.362,A -85,B 0,C 180,E1 -7434.727,E2 -7434.727} C_VEL
LIN {X 0,Y 474.636,Z 500.355,A -85,B 0,C 180,E1 -7437.789,E2 -7437.789} C_VEL
LIN {X 0,Y 474.626,Z 500.365,A -85,B 0,C 180,E1 -7440.885,E2 -7440.885} C_VEL
LIN {X 0,Y 474.727,Z 500.434,A -85,B 0,C 180,E1 -7443.307,E2 -7443.307} C_VEL
LIN {X 0,Y 476.549,Z 510.593,A -85,B 0,C 180,E1 -7445.147,E2 -7445.147} C_VEL
LIN {X 0,Y 476.329,Z 521.265,A -85,B 0,C 180,E1 -7446.984,E2 -7446.984} C_VEL
LIN {X 0,Y 475.961,Z 533.953,A -85,B 0,C 180,E1 -7449.137,E2 -7449.137} C_VEL
LIN {X 0,Y 475.2,Z 536.354,A -85,B 0,C 180,E1 -7449.51,E2 -7449.51} C_VEL
LIN {X 0,Y 469.331,Z 544.453,A -85,B 0,C 180,E1 -7450.617,E2 -7450.617} C_VEL
LIN {X 0,Y 468.732,Z 546.895,A -85,B 0,C 180,E1 -7450.992,E2 -7450.992} C_VEL
LIN {X 0,Y 469.125,Z 549.422,A -85,B 0,C 180,E1 -7451.082,E2 -7451.082} C_VEL
LIN {X 0,Y 471.4,Z 563.379,A -85,B 0,C 180,E1 -7451.389,E2 -7451.389} C_VEL
LIN {X 0,Y 470.599,Z 655.894,A -85,B 0,C 180,E1 -7452.828,E2 -7452.828} C_VEL
LIN {X 0,Y 470.343,Z 669.001,A -85,B 0,C 180,E1 -7453.196,E2 -7453.196} C_VEL
LIN {X 0,Y 469.992,Z 681.236,A -85,B 0,C 180,E1 -7453.718,E2 -7453.718} C_VEL
LIN {X 0,Y 469.522,Z 692.669,A -85,B 0,C 180,E1 -7454.37,E2 -7454.37} C_VEL
LIN {X 0,Y 469.015,Z 704.512,A -85,B 0,C 180,E1 -7455.242,E2 -7455.242} C_VEL
LIN {X 0,Y 468.447,Z 714.977,A -85,B 0,C 180,E1 -7456.222,E2 -7456.222} C_VEL
LIN {X 0,Y 468.027,Z 724.569,A -85,B 0,C 180,E1 -7457.333,E2 -7457.333} C_VEL
LIN {X 0,Y 467.679,Z 732.867,A -85,B 0,C 180,E1 -7458.515,E2 -7458.515} C_VEL
LIN {X 0,Y 467.236,Z 740.267,A -85,B 0,C 180,E1 -7459.82,E2 -7459.82} C_VEL
LIN {X 0,Y 466.986,Z 747.096,A -85,B 0,C 180,E1 -7461.344,E2 -7461.344} C_VEL
LIN {X 0,Y 466.84,Z 751.595,A -85,B 0,C 180,E1 -7462.648,E2 -7462.648} C_VEL
LIN {X 0,Y 466.756,Z 754.995,A -85,B 0,C 180,E1 -7463.95,E2 -7463.95} C_VEL
LIN {X 0,Y 466.709,Z 756.692,A -85,B 0,C 180,E1 -7464.816,E2 -7464.816} C_VEL
LIN {X 0,Y 466.673,Z 758.874,A -85,B 0,C 180,E1 -7466.547,E2 -7466.547} C_VEL
LIN {X 0,Y 466.659,Z 759.371,A -85,B 0,C 180,E1 -7467.411,E2 -7467.411} C_VEL
LIN {X 0,Y 466.62,Z 759.14,A -85,B 0,C 180,E1 -7469.137,E2 -7469.137} C_VEL
LIN {X 0,Y 466.601,Z 758.458,A -85,B 0,C 180,E1 -7470,E2 -7470} C_VEL
LIN {X 0,Y 466.626,Z 757.359,A -85,B 0,C 180,E1 -7470.863,E2 -7470.863} C_VEL
LIN {X 0,Y 466.721,Z 755.833,A -85,B 0,C 180,E1 -7471.726,E2 -7471.726} C_VEL
LIN {X 0,Y 466.861,Z 752.763,A -85,B 0,C 180,E1 -7473.02,E2 -7473.02} C_VEL
LIN {X 0,Y 466.996,Z 748.651,A -85,B 0,C 180,E1 -7474.315,E2 -7474.315} C_VEL
LIN {X 0,Y 467.143,Z 742.406,A -85,B 0,C 180,E1 -7475.828,E2 -7475.828} C_VEL
LIN {X 0,Y 467.538,Z 735.084,A -85,B 0,C 180,E1 -7477.199,E2 -7477.199} C_VEL
LIN {X 0,Y 467.893,Z 726.987,A -85,B 0,C 180,E1 -7478.421,E2 -7478.421} C_VEL
LIN {X 0,Y 468.348,Z 718.231,A -85,B 0,C 180,E1 -7479.501,E2 -7479.501} C_VEL
LIN {X 0,Y 468.859,Z 708.603,A -85,B 0,C 180,E1 -7480.471,E2 -7480.471} C_VEL
LIN {X 0,Y 469.301,Z 697.985,A -85,B 0,C 180,E1 -7481.335,E2 -7481.335} C_VEL
LIN {X 0,Y 469.712,Z 686.223,A -85,B 0,C 180,E1 -7482.091,E2 -7482.091} C_VEL
LIN {X 0,Y 470.208,Z 673.972,A -85,B 0,C 180,E1 -7482.681,E2 -7482.681} C_VEL
LIN {X 0,Y 470.463,Z 661.185,A -85,B 0,C 180,E1 -7483.113,E2 -7483.113} C_VEL
LIN {X 0,Y 470.668,Z 648.035,A -85,B 0,C 180,E1 -7483.382,E2 -7483.382} C_VEL
LIN {X 0,Y 471.239,Z 562.034,A -85,B 0,C 180,E1 -7484.699,E2 -7484.699} C_VEL
LIN {X 0,Y 468.675,Z 547.021,A -85,B 0,C 180,E1 -7485.046,E2 -7485.046} C_VEL
LIN {X 0,Y 469.076,Z 529.964,A -85,B 0,C 180,E1 -7487.887,E2 -7487.887} C_VEL
LIN {X 0,Y 469.68,Z 512.795,A -85,B 0,C 180,E1 -7490.816,E2 -7490.816} C_VEL
LIN {X 0,Y 467.6,Z 501.247,A -85,B 0,C 180,E1 -7492.944,E2 -7492.944} C_VEL
LIN {X 0,Y 467.613,Z 501.237,A -85,B 0,C 180,E1 -7495.839,E2 -7495.839} C_VEL
LIN {X 0,Y 467.579,Z 501.244,A -85,B 0,C 180,E1 -7498.749,E2 -7498.749} C_VEL
LIN {X 0,Y 467.585,Z 501.24,A -85,B 0,C 180,E1 -7501.739,E2 -7501.739} C_VEL
LIN {X 0,Y 467.565,Z 501.245,A -85,B 0,C 180,E1 -7504.832,E2 -7504.832} C_VEL
LIN {X 0,Y 467.565,Z 501.24,A -85,B 0,C 180,E1 -7508.043,E2 -7508.043} C_VEL
LIN {X 0,Y 467.581,Z 501.241,A -85,B 0,C 180,E1 -7511.276,E2 -7511.276} C_VEL
LIN {X 0,Y 467.572,Z 501.237,A -85,B 0,C 180,E1 -7513.822,E2 -7513.822} C_VEL
LIN {X 0,Y 467.573,Z 501.235,A -85,B 0,C 180,E1 -7516.257,E2 -7516.257} C_VEL
LIN {X 0,Y 467.578,Z 501.245,A -85,B 0,C 180,E1 -7518.722,E2 -7518.722} C_VEL
LIN {X 0,Y 467.562,Z 501.241,A -85,B 0,C 180,E1 -7521.955,E2 -7521.955} C_VEL
LIN {X 0,Y 467.564,Z 501.245,A -85,B 0,C 180,E1 -7525.167,E2 -7525.167} C_VEL
LIN {X 0,Y 467.646,Z 501.262,A -85,B 0,C 180,E1 -7526.668,E2 -7526.668} C_VEL
LIN {X 0,Y 467.947,Z 502.938,A -85,B 0,C 180,E1 -7527.086,E2 -7527.086} C_VEL
LIN {X 0,Y 470.546,Z 512.513,A -85,B 0,C 180,E1 -7527.344,E2 -7527.344} C_VEL
LIN {X 0,Y 471.345,Z 516.959,A -85,B 0,C 180,E1 -7527.448,E2 -7527.448} C_VEL
LIN {X 0,Y 470.37,Z 609.037,A -85,B 0,C 180,E1 -7528.97,E2 -7528.97} C_VEL
LIN {X 0,Y 470.099,Z 622.27,A -85,B 0,C 180,E1 -7529.355,E2 -7529.355} C_VEL
LIN {X 0,Y 469.889,Z 634.628,A -85,B 0,C 180,E1 -7529.89,E2 -7529.89} C_VEL
LIN {X 0,Y 469.473,Z 645.632,A -85,B 0,C 180,E1 -7530.518,E2 -7530.518} C_VEL
LIN {X 0,Y 469.016,Z 656.903,A -85,B 0,C 180,E1 -7531.346,E2 -7531.346} C_VEL
LIN {X 0,Y 468.575,Z 667.211,A -85,B 0,C 180,E1 -7532.292,E2 -7532.292} C_VEL
LIN {X 0,Y 468.208,Z 675.656,A -85,B 0,C 180,E1 -7533.236,E2 -7533.236} C_VEL
LIN {X 0,Y 467.836,Z 684.453,A -85,B 0,C 180,E1 -7534.428,E2 -7534.428} C_VEL
LIN {X 0,Y 467.453,Z 692.604,A -85,B 0,C 180,E1 -7535.814,E2 -7535.814} C_VEL
LIN {X 0,Y 467.233,Z 698.129,A -85,B 0,C 180,E1 -7536.978,E2 -7536.978} C_VEL
LIN {X 0,Y 467.029,Z 703.371,A -85,B 0,C 180,E1 -7538.365,E2 -7538.365} C_VEL
LIN {X 0,Y 466.874,Z 707.312,A -85,B 0,C 180,E1 -7539.743,E2 -7539.743} C_VEL
LIN {X 0,Y 466.766,Z 709.308,A -85,B 0,C 180,E1 -7540.655,E2 -7540.655} C_VEL
LIN {X 0,Y 466.742,Z 710.77,A -85,B 0,C 180,E1 -7541.566,E2 -7541.566} C_VEL
LIN {X 0,Y 466.681,Z 711.803,A -85,B 0,C 180,E1 -7542.471,E2 -7542.471} C_VEL
LIN {X 0,Y 466.669,Z 712.404,A -85,B 0,C 180,E1 -7543.373,E2 -7543.373} C_VEL
LIN {X 0,Y 466.703,Z 712.483,A -85,B 0,C 180,E1 -7544.524,E2 -7544.524} C_VEL
LIN {X 0,Y 466.706,Z 711.53,A -85,B 0,C 180,E1 -7546.058,E2 -7546.058} C_VEL
LIN {X 0,Y 466.761,Z 710.358,A -85,B 0,C 180,E1 -7546.947,E2 -7546.947} C_VEL
LIN {X 0,Y 466.885,Z 708.262,A -85,B 0,C 180,E1 -7548.075,E2 -7548.075} C_VEL
LIN {X 0,Y 467.031,Z 704.193,A -85,B 0,C 180,E1 -7549.596,E2 -7549.596} C_VEL
LIN {X 0,Y 467.255,Z 699.449,A -85,B 0,C 180,E1 -7550.913,E2 -7550.913} C_VEL
LIN {X 0,Y 467.499,Z 693.446,A -85,B 0,C 180,E1 -7552.224,E2 -7552.224} C_VEL
LIN {X 0,Y 467.856,Z 685.956,A -85,B 0,C 180,E1 -7553.531,E2 -7553.531} C_VEL
LIN {X 0,Y 468.18,Z 678.317,A -85,B 0,C 180,E1 -7554.616,E2 -7554.616} C_VEL
LIN {X 0,Y 468.628,Z 667.945,A -85,B 0,C 180,E1 -7555.807,E2 -7555.807} C_VEL
LIN {X 0,Y 469.078,Z 657.405,A -85,B 0,C 180,E1 -7556.779,E2 -7556.779} C_VEL
LIN {X 0,Y 469.485,Z 647.223,A -85,B 0,C 180,E1 -7557.533,E2 -7557.533} C_VEL
LIN {X 0,Y 469.925,Z 635.062,A -85,B 0,C 180,E1 -7558.232,E2 -7558.232} C_VEL
LIN {X 0,Y 470.228,Z 621.717,A -85,B 0,C 180,E1 -7558.795,E2 -7558.795} C_VEL
LIN {X 0,Y 470.434,Z 609.255,A -85,B 0,C 180,E1 -7559.144,E2 -7559.144} C_VEL
LIN {X 0,Y 471.425,Z 516.071,A -85,B 0,C 180,E1 -7560.721,E2 -7560.721} C_VEL
LIN {X 0,Y 468.629,Z 505.646,A -85,B 0,C 180,E1 -7561.02,E2 -7561.02} C_VEL
LIN {X 0,Y 468.486,Z 505.125,A -85,B 0,C 180,E1 -7561.074,E2 -7561.074} C_VEL
LIN {X 0,Y 467.771,Z 501.22,A -85,B 0,C 180,E1 -7562.152,E2 -7562.152} C_VEL
LIN {X 0,Y 467.745,Z 501.221,A -85,B 0,C 180,E1 -7566.037,E2 -7566.037} C_VEL
LIN {X 0,Y 467.673,Z 501.23,A -85,B 0,C 180,E1 -7568.643,E2 -7568.643} C_VEL
LIN {X 0,Y 467.681,Z 501.226,A -85,B 0,C 180,E1 -7572.379,E2 -7572.379} C_VEL
LIN {X 0,Y 467.64,Z 501.232,A -85,B 0,C 180,E1 -7575.886,E2 -7575.886} C_VEL
LIN {X 0,Y 467.615,Z 501.239,A -85,B 0,C 180,E1 -7579.308,E2 -7579.308} C_VEL
LIN {X 0,Y 467.527,Z 501.245,A -85,B 0,C 180,E1 -7582.074,E2 -7582.074} C_VEL
LIN {X 0,Y 467.595,Z 501.24,A -85,B 0,C 180,E1 -7584.888,E2 -7584.888} C_VEL
LIN {X 0,Y 467.62,Z 501.231,A -85,B 0,C 180,E1 -7587.769,E2 -7587.769} C_VEL
LIN {X 0,Y 467.565,Z 501.244,A -85,B 0,C 180,E1 -7591.046,E2 -7591.046} C_VEL
LIN {X 0,Y 467.583,Z 501.235,A -85,B 0,C 180,E1 -7594.243,E2 -7594.243} C_VEL
LIN {X 0,Y 467.544,Z 501.247,A -85,B 0,C 180,E1 -7597.187,E2 -7597.187} C_VEL
LIN {X 0,Y 467.572,Z 501.239,A -85,B 0,C 180,E1 -7600.265,E2 -7600.265} C_VEL
LIN {X 0,Y 467.581,Z 501.24,A -85,B 0,C 180,E1 -7602.568,E2 -7602.568} C_VEL
LIN {X 0,Y 467.566,Z 501.246,A -85,B 0,C 180,E1 -7605.054,E2 -7605.054} C_VEL
LIN {X 0,Y 467.585,Z 501.242,A -85,B 0,C 180,E1 -7607.441,E2 -7607.441} C_VEL
LIN {X 0,Y 467.579,Z 501.245,A -85,B 0,C 180,E1 -7610.856,E2 -7610.856} C_VEL
LIN {X 0,Y 467.56,Z 501.243,A -85,B 0,C 180,E1 -7614.261,E2 -7614.261} C_VEL
LIN {X 0,Y 467.581,Z 501.246,A -85,B 0,C 180,E1 -7617.321,E2 -7617.321} C_VEL
LIN {X 0,Y 467.569,Z 501.246,A -85,B 0,C 180,E1 -7620.668,E2 -7620.668} C_VEL
LIN {X 0,Y 467.65,Z 501.406,A -85,B 0,C 180,E1 -7622.112,E2 -7622.112} C_VEL
LIN {X 0,Y 470.179,Z 513.726,A -85,B 0,C 180,E1 -7624.312,E2 -7624.312} C_VEL
LIN {X 0,Y 470.383,Z 518.069,A -85,B 0,C 180,E1 -7625.034,E2 -7625.034} C_VEL
LIN {X 0,Y 469.366,Z 540.141,A -85,B 0,C 180,E1 -7628.529,E2 -7628.529} C_VEL
LIN {X 0,Y 468.601,Z 560.201,A -85,B 0,C 180,E1 -7631.642,E2 -7631.642} C_VEL
LIN {X 0,Y 468.293,Z 568.676,A -85,B 0,C 180,E1 -7632.941,E2 -7632.941} C_VEL
LIN {X 0,Y 471.101,Z 591.126,A -85,B 0,C 180,E1 -7633.442,E2 -7633.442} C_VEL
LIN {X 0,Y 470.211,Z 679.118,A -85,B 0,C 180,E1 -7634.921,E2 -7634.921} C_VEL
LIN {X 0,Y 469.799,Z 692.814,A -85,B 0,C 180,E1 -7635.323,E2 -7635.323} C_VEL
LIN {X 0,Y 469.332,Z 707.071,A -85,B 0,C 180,E1 -7635.917,E2 -7635.917} C_VEL
LIN {X 0,Y 468.903,Z 718.546,A -85,B 0,C 180,E1 -7636.567,E2 -7636.567} C_VEL
LIN {X 0,Y 468.493,Z 730.369,A -85,B 0,C 180,E1 -7637.446,E2 -7637.446} C_VEL
LIN {X 0,Y 468.024,Z 740.735,A -85,B 0,C 180,E1 -7638.414,E2 -7638.414} C_VEL
LIN {X 0,Y 467.63,Z 749.284,A -85,B 0,C 180,E1 -7639.391,E2 -7639.391} C_VEL
LIN {X 0,Y 467.322,Z 757.146,A -85,B 0,C 180,E1 -7640.478,E2 -7640.478} C_VEL
LIN {X 0,Y 467.053,Z 764.782,A -85,B 0,C 180,E1 -7641.782,E2 -7641.782} C_VEL
LIN {X 0,Y 466.856,Z 770.898,A -85,B 0,C 180,E1 -7643.083,E2 -7643.083} C_VEL
LIN {X 0,Y 466.823,Z 775.73,A -85,B 0,C 180,E1 -7644.384,E2 -7644.384} C_VEL
LIN {X 0,Y 466.706,Z 779.417,A -85,B 0,C 180,E1 -7645.682,E2 -7645.682} C_VEL
LIN {X 0,Y 466.711,Z 781.316,A -85,B 0,C 180,E1 -7646.547,E2 -7646.547} C_VEL
LIN {X 0,Y 466.746,Z 782.751,A -85,B 0,C 180,E1 -7647.411,E2 -7647.411} C_VEL
LIN {X 0,Y 466.628,Z 784.374,A -85,B 0,C 180,E1 -7649.137,E2 -7649.137} C_VEL
LIN {X 0,Y 466.615,Z 784.595,A -85,B 0,C 180,E1 -7650,E2 -7650} C_VEL
LIN {X 0,Y 466.627,Z 784.373,A -85,B 0,C 180,E1 -7650.863,E2 -7650.863} C_VEL
LIN {X 0,Y 466.747,Z 782.747,A -85,B 0,C 180,E1 -7652.589,E2 -7652.589} C_VEL
LIN {X 0,Y 466.722,Z 781.312,A -85,B 0,C 180,E1 -7653.453,E2 -7653.453} C_VEL
LIN {X 0,Y 466.706,Z 778.326,A -85,B 0,C 180,E1 -7654.751,E2 -7654.751} C_VEL
LIN {X 0,Y 466.794,Z 774.275,A -85,B 0,C 180,E1 -7656.05,E2 -7656.05} C_VEL
LIN {X 0,Y 466.943,Z 768.016,A -85,B 0,C 180,E1 -7657.567,E2 -7657.567} C_VEL
LIN {X 0,Y 467.147,Z 761.186,A -85,B 0,C 180,E1 -7658.871,E2 -7658.871} C_VEL
LIN {X 0,Y 467.402,Z 754.206,A -85,B 0,C 180,E1 -7659.957,E2 -7659.957} C_VEL
LIN {X 0,Y 467.786,Z 745.77,A -85,B 0,C 180,E1 -7661.043,E2 -7661.043} C_VEL
LIN {X 0,Y 468.216,Z 735.304,A -85,B 0,C 180,E1 -7662.13,E2 -7662.13} C_VEL
LIN {X 0,Y 468.693,Z 724.919,A -85,B 0,C 180,E1 -7662.998,E2 -7662.998} C_VEL
LIN {X 0,Y 469.115,Z 713.459,A -85,B 0,C 180,E1 -7663.758,E2 -7663.758} C_VEL
LIN {X 0,Y 469.594,Z 700.873,A -85,B 0,C 180,E1 -7664.407,E2 -7664.407} C_VEL
LIN {X 0,Y 470.027,Z 687.776,A -85,B 0,C 180,E1 -7664.891,E2 -7664.891} C_VEL
LIN {X 0,Y 470.356,Z 673.86,A -85,B 0,C 180,E1 -7665.213,E2 -7665.213} C_VEL
LIN {X 0,Y 470.975,Z 589.422,A -85,B 0,C 180,E1 -7666.598,E2 -7666.598} C_VEL
LIN {X 0,Y 468.421,Z 570.531,A -85,B 0,C 180,E1 -7667.012,E2 -7667.012} C_VEL
LIN {X 0,Y 469.22,Z 550.216,A -85,B 0,C 180,E1 -7670.15,E2 -7670.15} C_VEL
LIN {X 0,Y 469.993,Z 531.271,A -85,B 0,C 180,E1 -7673.111,E2 -7673.111} C_VEL
LIN {X 0,Y 470.675,Z 516.686,A -85,B 0,C 180,E1 -7675.422,E2 -7675.422} C_VEL
LIN {X 0,Y 468.36,Z 504.629,A -85,B 0,C 180,E1 -7677.503,E2 -7677.503} C_VEL
LIN {X 0,Y 467.62,Z 501.237,A -85,B 0,C 180,E1 -7678.134,E2 -7678.134} C_VEL
LIN {X 0,Y 467.582,Z 501.241,A -85,B 0,C 180,E1 -7681.739,E2 -7681.739} C_VEL
LIN {X 0,Y 467.562,Z 501.244,A -85,B 0,C 180,E1 -7684.832,E2 -7684.832} C_VEL
LIN {X 0,Y 467.562,Z 501.222,A -85,B 0,C 180,E1 -7688.044,E2 -7688.044} C_VEL
LIN {X 0,Y 467.578,Z 501.245,A -85,B 0,C 180,E1 -7691.277,E2 -7691.277} C_VEL
LIN {X 0,Y 467.569,Z 501.237,A -85,B 0,C 180,E1 -7693.823,E2 -7693.823} C_VEL
LIN {X 0,Y 467.551,Z 501.242,A -85,B 0,C 180,E1 -7696.255,E2 -7696.255} C_VEL
LIN {X 0,Y 467.579,Z 501.235,A -85,B 0,C 180,E1 -7698.722,E2 -7698.722} C_VEL
LIN {X 0,Y 467.567,Z 501.242,A -85,B 0,C 180,E1 -7701.407,E2 -7701.407} C_VEL
LIN {X 0,Y 467.556,Z 501.236,A -85,B 0,C 180,E1 -7704.26,E2 -7704.26} C_VEL
LIN {X 0,Y 467.575,Z 501.24,A -85,B 0,C 180,E1 -7707.32,E2 -7707.32} C_VEL
LIN {X 0,Y 467.57,Z 501.235,A -85,B 0,C 180,E1 -7710.665,E2 -7710.665} C_VEL
LIN {X 0,Y 467.62,Z 501.237,A -85,B 0,C 180,E1 -7713.2,E2 -7713.2} C_VEL
LIN {X 0,Y 467.584,Z 501.226,A -85,B 0,C 180,E1 -7716.468,E2 -7716.468} C_VEL
LIN {X 0,Y 467.615,Z 501.233,A -85,B 0,C 180,E1 -7719.777,E2 -7719.777} C_VEL
LIN {X 0,Y 467.6,Z 501.23,A -85,B 0,C 180,E1 -7722.507,E2 -7722.507} C_VEL
LIN {X 0,Y 467.597,Z 501.235,A -85,B 0,C 180,E1 -7725.196,E2 -7725.196} C_VEL
LIN {X 0,Y 467.674,Z 501.226,A -85,B 0,C 180,E1 -7727.855,E2 -7727.855} C_VEL
LIN {X 0,Y 467.673,Z 501.218,A -85,B 0,C 180,E1 -7731.357,E2 -7731.357} C_VEL
LIN {X 0,Y 467.744,Z 501.214,A -85,B 0,C 180,E1 -7733.963,E2 -7733.963} C_VEL
LIN {X 0,Y 467.851,Z 501.203,A -85,B 0,C 180,E1 -7737.417,E2 -7737.417} C_VEL
LIN {X 0,Y 467.873,Z 501.186,A -85,B 0,C 180,E1 -7740,E2 -7740} C_VEL
LIN {X 0,Y 467.852,Z 501.201,A -85,B 0,C 180,E1 -7742.583,E2 -7742.583} C_VEL
LIN {X 0,Y 467.745,Z 501.214,A -85,B 0,C 180,E1 -7746.038,E2 -7746.038} C_VEL
LIN {X 0,Y 467.674,Z 501.216,A -85,B 0,C 180,E1 -7748.643,E2 -7748.643} C_VEL
LIN {X 0,Y 467.648,Z 501.229,A -85,B 0,C 180,E1 -7752.146,E2 -7752.146} C_VEL
LIN {X 0,Y 467.63,Z 501.221,A -85,B 0,C 180,E1 -7755.696,E2 -7755.696} C_VEL
LIN {X 0,Y 467.61,Z 501.235,A -85,B 0,C 180,E1 -7758.765,E2 -7758.765} C_VEL
LIN {X 0,Y 467.573,Z 501.239,A -85,B 0,C 180,E1 -7761.269,E2 -7761.269} C_VEL
LIN {X 0,Y 467.565,Z 501.233,A -85,B 0,C 180,E1 -7763.944,E2 -7763.944} C_VEL
LIN {X 0,Y 467.621,Z 501.237,A -85,B 0,C 180,E1 -7766.8,E2 -7766.8} C_VEL
LIN {X 0,Y 467.583,Z 501.232,A -85,B 0,C 180,E1 -7769.737,E2 -7769.737} C_VEL
LIN {X 0,Y 467.578,Z 501.242,A -85,B 0,C 180,E1 -7772.759,E2 -7772.759} C_VEL
LIN {X 0,Y 467.553,Z 501.24,A -85,B 0,C 180,E1 -7775.89,E2 -7775.89} C_VEL
LIN {X 0,Y 467.579,Z 501.241,A -85,B 0,C 180,E1 -7779.146,E2 -7779.146} C_VEL
LIN {X 0,Y 467.583,Z 501.242,A -85,B 0,C 180,E1 -7782.568,E2 -7782.568} C_VEL
LIN {X 0,Y 467.569,Z 501.248,A -85,B 0,C 180,E1 -7785.054,E2 -7785.054} C_VEL
LIN {X 0,Y 467.587,Z 501.24,A -85,B 0,C 180,E1 -7787.441,E2 -7787.441} C_VEL
LIN {X 0,Y 467.582,Z 501.243,A -85,B 0,C 180,E1 -7790.856,E2 -7790.856} C_VEL
LIN {X 0,Y 467.559,Z 501.241,A -85,B 0,C 180,E1 -7794.262,E2 -7794.262} C_VEL
LIN {X 0,Y 467.582,Z 501.238,A -85,B 0,C 180,E1 -7797.322,E2 -7797.322} C_VEL
LIN {X 0,Y 467.572,Z 501.242,A -85,B 0,C 180,E1 -7800.668,E2 -7800.668} C_VEL
LIN {X 0,Y 467.685,Z 501.252,A -85,B 0,C 180,E1 -7803.093,E2 -7803.093} C_VEL
LIN {X 0,Y 469.58,Z 511.594,A -85,B 0,C 180,E1 -7804.989,E2 -7804.989} C_VEL
LIN {X 0,Y 469.41,Z 522.353,A -85,B 0,C 180,E1 -7806.858,E2 -7806.858} C_VEL
LIN {X 0,Y 468.844,Z 539.843,A -85,B 0,C 180,E1 -7809.833,E2 -7809.833} C_VEL
LIN {X 0,Y 468.732,Z 546.895,A -85,B 0,C 180,E1 -7810.992,E2 -7810.992} C_VEL
LIN {X 0,Y 468.371,Z 548.216,A -85,B 0,C 180,E1 -7811.034,E2 -7811.034} C_VEL
LIN {X 0,Y 464.244,Z 562.088,A -85,B 0,C 180,E1 -7811.076,E2 -7811.076} C_VEL
LIN {X 0,Y 464.023,Z 567.483,A -85,B 0,C 180,E1 -7811.124,E2 -7811.124} C_VEL
LIN {X 0,Y 464.499,Z 578.287,A -85,B 0,C 180,E1 -7811.361,E2 -7811.361} C_VEL
LIN {X 0,Y 463.75,Z 656.74,A -85,B 0,C 180,E1 -7812.606,E2 -7812.606} C_VEL
LIN {X 0,Y 463.486,Z 669.418,A -85,B 0,C 180,E1 -7812.973,E2 -7812.973} C_VEL
LIN {X 0,Y 463.115,Z 682.02,A -85,B 0,C 180,E1 -7813.526,E2 -7813.526} C_VEL
LIN {X 0,Y 462.605,Z 694.175,A -85,B 0,C 180,E1 -7814.243,E2 -7814.243} C_VEL
LIN {X 0,Y 462.055,Z 705.682,A -85,B 0,C 180,E1 -7815.128,E2 -7815.128} C_VEL
LIN {X 0,Y 461.404,Z 717.012,A -85,B 0,C 180,E1 -7816.232,E2 -7816.232} C_VEL
LIN {X 0,Y 461.007,Z 726.092,A -85,B 0,C 180,E1 -7817.339,E2 -7817.339} C_VEL
LIN {X 0,Y 460.608,Z 734.234,A -85,B 0,C 180,E1 -7818.559,E2 -7818.559} C_VEL
LIN {X 0,Y 460.174,Z 741.427,A -85,B 0,C 180,E1 -7819.885,E2 -7819.885} C_VEL
LIN {X 0,Y 459.921,Z 747.187,A -85,B 0,C 180,E1 -7821.21,E2 -7821.21} C_VEL
LIN {X 0,Y 459.782,Z 751.708,A -85,B 0,C 180,E1 -7822.535,E2 -7822.535} C_VEL
LIN {X 0,Y 459.67,Z 755.129,A -85,B 0,C 180,E1 -7823.856,E2 -7823.856} C_VEL
LIN {X 0,Y 459.644,Z 756.842,A -85,B 0,C 180,E1 -7824.736,E2 -7824.736} C_VEL
LIN {X 0,Y 459.57,Z 759.043,A -85,B 0,C 180,E1 -7826.493,E2 -7826.493} C_VEL
LIN {X 0,Y 459.581,Z 759.555,A -85,B 0,C 180,E1 -7827.371,E2 -7827.371} C_VEL
LIN {X 0,Y 459.524,Z 759.344,A -85,B 0,C 180,E1 -7829.124,E2 -7829.124} C_VEL
LIN {X 0,Y 459.533,Z 758.67,A -85,B 0,C 180,E1 -7830,E2 -7830} C_VEL
LIN {X 0,Y 459.531,Z 757.589,A -85,B 0,C 180,E1 -7830.876,E2 -7830.876} C_VEL
LIN {X 0,Y 459.628,Z 756.072,A -85,B 0,C 180,E1 -7831.752,E2 -7831.752} C_VEL
LIN {X 0,Y 459.776,Z 753.02,A -85,B 0,C 180,E1 -7833.067,E2 -7833.067} C_VEL
LIN {X 0,Y 459.915,Z 748.927,A -85,B 0,C 180,E1 -7834.382,E2 -7834.382} C_VEL
LIN {X 0,Y 460.098,Z 742.7,A -85,B 0,C 180,E1 -7835.918,E2 -7835.918} C_VEL
LIN {X 0,Y 460.512,Z 735.734,A -85,B 0,C 180,E1 -7837.256,E2 -7837.256} C_VEL
LIN {X 0,Y 460.9,Z 727.338,A -85,B 0,C 180,E1 -7838.55,E2 -7838.55} C_VEL
LIN {X 0,Y 461.368,Z 718.611,A -85,B 0,C 180,E1 -7839.646,E2 -7839.646} C_VEL
LIN {X 0,Y 461.91,Z 709.032,A -85,B 0,C 180,E1 -7840.631,E2 -7840.631} C_VEL
LIN {X 0,Y 462.364,Z 698.468,A -85,B 0,C 180,E1 -7841.508,E2 -7841.508} C_VEL
LIN {X 0,Y 462.797,Z 686.771,A -85,B 0,C 180,E1 -7842.275,E2 -7842.275} C_VEL
LIN {X 0,Y 463.319,Z 674.676,A -85,B 0,C 180,E1 -7842.873,E2 -7842.873} C_VEL
LIN {X 0,Y 463.591,Z 662.12,A -85,B 0,C 180,E1 -7843.311,E2 -7843.311} C_VEL
LIN {X 0,Y 463.808,Z 649.538,A -85,B 0,C 180,E1 -7843.584,E2 -7843.584} C_VEL
LIN {X 0,Y 464.434,Z 562.921,A -85,B 0,C 180,E1 -7844.929,E2 -7844.929} C_VEL
LIN {X 0,Y 461.754,Z 547.268,A -85,B 0,C 180,E1 -7845.277,E2 -7845.277} C_VEL
LIN {X 0,Y 462.177,Z 530.048,A -85,B 0,C 180,E1 -7848.163,E2 -7848.163} C_VEL
LIN {X 0,Y 462.746,Z 514.059,A -85,B 0,C 180,E1 -7850.91,E2 -7850.91} C_VEL
LIN {X 0,Y 460.556,Z 502.125,A -85,B 0,C 180,E1 -7853.137,E2 -7853.137} C_VEL
LIN {X 0,Y 460.566,Z 502.115,A -85,B 0,C 180,E1 -7856.264,E2 -7856.264} C_VEL
LIN {X 0,Y 460.542,Z 502.121,A -85,B 0,C 180,E1 -7859.23,E2 -7859.23} C_VEL
LIN {X 0,Y 460.533,Z 502.118,A -85,B 0,C 180,E1 -7862.283,E2 -7862.283} C_VEL
LIN {X 0,Y 460.511,Z 502.12,A -85,B 0,C 180,E1 -7865.445,E2 -7865.445} C_VEL
LIN {X 0,Y 460.544,Z 502.12,A -85,B 0,C 180,E1 -7868.897,E2 -7868.897} C_VEL
LIN {X 0,Y 460.524,Z 502.117,A -85,B 0,C 180,E1 -7872.18,E2 -7872.18} C_VEL
LIN {X 0,Y 460.519,Z 502.114,A -85,B 0,C 180,E1 -7875.411,E2 -7875.411} C_VEL
LIN {X 0,Y 460.532,Z 502.118,A -85,B 0,C 180,E1 -7878.396,E2 -7878.396} C_VEL
LIN {X 0,Y 460.523,Z 502.12,A -85,B 0,C 180,E1 -7881.266,E2 -7881.266} C_VEL
LIN {X 0,Y 460.509,Z 502.125,A -85,B 0,C 180,E1 -7884.554,E2 -7884.554} C_VEL
LIN {X 0,Y 460.643,Z 502.274,A -85,B 0,C 180,E1 -7886.553,E2 -7886.553} C_VEL
LIN {X 0,Y 460.882,Z 503.517,A -85,B 0,C 180,E1 -7886.831,E2 -7886.831} C_VEL
LIN {X 0,Y 463.471,Z 512.44,A -85,B 0,C 180,E1 -7887.085,E2 -7887.085} C_VEL
LIN {X 0,Y 464.503,Z 517.222,A -85,B 0,C 180,E1 -7887.206,E2 -7887.206} C_VEL
LIN {X 0,Y 463.487,Z 610.03,A -85,B 0,C 180,E1 -7888.775,E2 -7888.775} C_VEL
LIN {X 0,Y 463.206,Z 623.926,A -85,B 0,C 180,E1 -7889.198,E2 -7889.198} C_VEL
LIN {X 0,Y 462.95,Z 636.125,A -85,B 0,C 180,E1 -7889.747,E2 -7889.747} C_VEL
LIN {X 0,Y 462.497,Z 647.164,A -85,B 0,C 180,E1 -7890.405,E2 -7890.405} C_VEL
LIN {X 0,Y 462.04,Z 658.242,A -85,B 0,C 180,E1 -7891.246,E2 -7891.246} C_VEL
LIN {X 0,Y 461.591,Z 668.505,A -85,B 0,C 180,E1 -7892.215,E2 -7892.215} C_VEL
LIN {X 0,Y 461.165,Z 677.717,A -85,B 0,C 180,E1 -7893.283,E2 -7893.283} C_VEL
LIN {X 0,Y 460.79,Z 685.698,A -85,B 0,C 180,E1 -7894.415,E2 -7894.415} C_VEL
LIN {X 0,Y 460.431,Z 692.891,A -85,B 0,C 180,E1 -7895.661,E2 -7895.661} C_VEL
LIN {X 0,Y 460.147,Z 699.45,A -85,B 0,C 180,E1 -7897.078,E2 -7897.078} C_VEL
LIN {X 0,Y 459.965,Z 704.536,A -85,B 0,C 180,E1 -7898.487,E2 -7898.487} C_VEL
LIN {X 0,Y 459.8,Z 708.321,A -85,B 0,C 180,E1 -7899.884,E2 -7899.884} C_VEL
LIN {X 0,Y 459.667,Z 711.16,A -85,B 0,C 180,E1 -7901.426,E2 -7901.426} C_VEL
LIN {X 0,Y 459.588,Z 712.804,A -85,B 0,C 180,E1 -7903.109,E2 -7903.109} C_VEL
LIN {X 0,Y 459.62,Z 713.047,A -85,B 0,C 180,E1 -7904.43,E2 -7904.43} C_VEL
LIN {X 0,Y 459.618,Z 712.304,A -85,B 0,C 180,E1 -7905.838,E2 -7905.838} C_VEL
LIN {X 0,Y 459.691,Z 711.288,A -85,B 0,C 180,E1 -7906.742,E2 -7906.742} C_VEL
LIN {X 0,Y 459.815,Z 709.075,A -85,B 0,C 180,E1 -7908.009,E2 -7908.009} C_VEL
LIN {X 0,Y 459.964,Z 705.502,A -85,B 0,C 180,E1 -7909.435,E2 -7909.435} C_VEL
LIN {X 0,Y 460.166,Z 700.991,A -85,B 0,C 180,E1 -7910.772,E2 -7910.772} C_VEL
LIN {X 0,Y 460.468,Z 695.225,A -85,B 0,C 180,E1 -7912.104,E2 -7912.104} C_VEL
LIN {X 0,Y 460.809,Z 688.009,A -85,B 0,C 180,E1 -7913.432,E2 -7913.432} C_VEL
LIN {X 0,Y 461.207,Z 679.066,A -85,B 0,C 180,E1 -7914.754,E2 -7914.754} C_VEL
LIN {X 0,Y 461.647,Z 669.799,A -85,B 0,C 180,E1 -7915.853,E2 -7915.853} C_VEL
LIN {X 0,Y 462.09,Z 659.523,A -85,B 0,C 180,E1 -7916.839,E2 -7916.839} C_VEL
LIN {X 0,Y 462.602,Z 648.101,A -85,B 0,C 180,E1 -7917.714,E2 -7917.714} C_VEL
LIN {X 0,Y 463.063,Z 636.053,A -85,B 0,C 180,E1 -7918.423,E2 -7918.423} C_VEL
LIN {X 0,Y 463.385,Z 622.849,A -85,B 0,C 180,E1 -7918.995,E2 -7918.995} C_VEL
LIN {X 0,Y 463.603,Z 609.798,A -85,B 0,C 180,E1 -7919.37,E2 -7919.37} C_VEL
LIN {X 0,Y 464.736,Z 517.383,A -85,B 0,C 180,E1 -7920.971,E2 -7920.971} C_VEL
LIN {X 0,Y 462.249,Z 508.256,A -85,B 0,C 180,E1 -7921.248,E2 -7921.248} C_VEL
LIN {X 0,Y 461.405,Z 505.944,A -85,B 0,C 180,E1 -7921.337,E2 -7921.337} C_VEL
LIN {X 0,Y 460.774,Z 502.091,A -85,B 0,C 180,E1 -7922.404,E2 -7922.404} C_VEL
LIN {X 0,Y 460.709,Z 502.097,A -85,B 0,C 180,E1 -7926.13,E2 -7926.13} C_VEL
LIN {X 0,Y 460.621,Z 502.109,A -85,B 0,C 180,E1 -7928.776,E2 -7928.776} C_VEL
LIN {X 0,Y 460.625,Z 502.106,A -85,B 0,C 180,E1 -7932.457,E2 -7932.457} C_VEL
LIN {X 0,Y 460.591,Z 502.11,A -85,B 0,C 180,E1 -7935.998,E2 -7935.998} C_VEL
LIN {X 0,Y 460.562,Z 502.116,A -85,B 0,C 180,E1 -7938.902,E2 -7938.902} C_VEL
LIN {X 0,Y 460.507,Z 502.122,A -85,B 0,C 180,E1 -7941.486,E2 -7941.486} C_VEL
LIN {X 0,Y 460.534,Z 502.115,A -85,B 0,C 180,E1 -7944.333,E2 -7944.333} C_VEL
LIN {X 0,Y 460.576,Z 502.113,A -85,B 0,C 180,E1 -7947.244,E2 -7947.244} C_VEL
LIN {X 0,Y 460.52,Z 502.115,A -85,B 0,C 180,E1 -7950.239,E2 -7950.239} C_VEL
LIN {X 0,Y 460.522,Z 502.118,A -85,B 0,C 180,E1 -7953.325,E2 -7953.325} C_VEL
LIN {X 0,Y 460.473,Z 502.122,A -85,B 0,C 180,E1 -7956.53,E2 -7956.53} C_VEL
LIN {X 0,Y 460.543,Z 502.119,A -85,B 0,C 180,E1 -7958.899,E2 -7958.899} C_VEL
LIN {X 0,Y 460.517,Z 502.117,A -85,B 0,C 180,E1 -7962.182,E2 -7962.182} C_VEL
LIN {X 0,Y 460.516,Z 502.121,A -85,B 0,C 180,E1 -7965.413,E2 -7965.413} C_VEL
LIN {X 0,Y 460.531,Z 502.12,A -85,B 0,C 180,E1 -7968.398,E2 -7968.398} C_VEL
LIN {X 0,Y 460.524,Z 502.121,A -85,B 0,C 180,E1 -7971.268,E2 -7971.268} C_VEL
LIN {X 0,Y 460.51,Z 502.124,A -85,B 0,C 180,E1 -7974.555,E2 -7974.555} C_VEL
LIN {X 0,Y 460.531,Z 502.122,A -85,B 0,C 180,E1 -7977.716,E2 -7977.716} C_VEL
LIN {X 0,Y 460.539,Z 502.122,A -85,B 0,C 180,E1 -7980.77,E2 -7980.77} C_VEL
LIN {X 0,Y 460.609,Z 502.272,A -85,B 0,C 180,E1 -7981.837,E2 -7981.837} C_VEL
LIN {X 0,Y 463.207,Z 514.824,A -85,B 0,C 180,E1 -7984.138,E2 -7984.138} C_VEL
LIN {X 0,Y 463.478,Z 519.167,A -85,B 0,C 180,E1 -7984.876,E2 -7984.876} C_VEL
LIN {X 0,Y 462.468,Z 540.193,A -85,B 0,C 180,E1 -7988.275,E2 -7988.275} C_VEL
LIN {X 0,Y 461.58,Z 561.144,A -85,B 0,C 180,E1 -7991.583,E2 -7991.583} C_VEL
LIN {X 0,Y 461.338,Z 567.995,A -85,B 0,C 180,E1 -7992.653,E2 -7992.653} C_VEL
LIN {X 0,Y 464.312,Z 591.971,A -85,B 0,C 180,E1 -7993.209,E2 -7993.209} C_VEL
LIN {X 0,Y 463.351,Z 678.437,A -85,B 0,C 180,E1 -7994.692,E2 -7994.692} C_VEL
LIN {X 0,Y 462.899,Z 692.987,A -85,B 0,C 180,E1 -7995.127,E2 -7995.127} C_VEL
LIN {X 0,Y 462.486,Z 705.643,A -85,B 0,C 180,E1 -7995.648,E2 -7995.648} C_VEL
LIN {X 0,Y 461.983,Z 718.271,A -85,B 0,C 180,E1 -7996.362,E2 -7996.362} C_VEL
LIN {X 0,Y 461.584,Z 729.596,A -85,B 0,C 180,E1 -7997.21,E2 -7997.21} C_VEL
LIN {X 0,Y 461.009,Z 740.491,A -85,B 0,C 180,E1 -7998.235,E2 -7998.235} C_VEL
LIN {X 0,Y 460.618,Z 749.052,A -85,B 0,C 180,E1 -7999.228,E2 -7999.228} C_VEL
LIN {X 0,Y 460.283,Z 756.923,A -85,B 0,C 180,E1 -8000.331,E2 -8000.331} C_VEL
LIN {X 0,Y 459.992,Z 764.567,A -85,B 0,C 180,E1 -8001.654,E2 -8001.654} C_VEL
LIN {X 0,Y 459.774,Z 770.689,A -85,B 0,C 180,E1 -8002.976,E2 -8002.976} C_VEL
LIN {X 0,Y 459.738,Z 775.526,A -85,B 0,C 180,E1 -8004.298,E2 -8004.298} C_VEL
LIN {X 0,Y 459.615,Z 779.217,A -85,B 0,C 180,E1 -8005.615,E2 -8005.615} C_VEL
LIN {X 0,Y 459.609,Z 781.117,A -85,B 0,C 180,E1 -8006.493,E2 -8006.493} C_VEL
LIN {X 0,Y 459.661,Z 782.555,A -85,B 0,C 180,E1 -8007.371,E2 -8007.371} C_VEL
LIN {X 0,Y 459.531,Z 784.181,A -85,B 0,C 180,E1 -8009.124,E2 -8009.124} C_VEL
LIN {X 0,Y 459.545,Z 784.405,A -85,B 0,C 180,E1 -8010,E2 -8010} C_VEL
LIN {X 0,Y 459.577,Z 783.568,A -85,B 0,C 180,E1 -8011.753,E2 -8011.753} C_VEL
LIN {X 0,Y 459.662,Z 782.561,A -85,B 0,C 180,E1 -8012.629,E2 -8012.629} C_VEL
LIN {X 0,Y 459.618,Z 781.129,A -85,B 0,C 180,E1 -8013.507,E2 -8013.507} C_VEL
LIN {X 0,Y 459.637,Z 778.149,A -85,B 0,C 180,E1 -8014.824,E2 -8014.824} C_VEL
LIN {X 0,Y 459.711,Z 774.103,A -85,B 0,C 180,E1 -8016.143,E2 -8016.143} C_VEL
LIN {X 0,Y 459.881,Z 767.852,A -85,B 0,C 180,E1 -8017.684,E2 -8017.684} C_VEL
LIN {X 0,Y 460.092,Z 761.031,A -85,B 0,C 180,E1 -8019.008,E2 -8019.008} C_VEL
LIN {X 0,Y 460.375,Z 754.062,A -85,B 0,C 180,E1 -8020.111,E2 -8020.111} C_VEL
LIN {X 0,Y 460.794,Z 745.643,A -85,B 0,C 180,E1 -8021.213,E2 -8021.213} C_VEL
LIN {X 0,Y 461.257,Z 735.198,A -85,B 0,C 180,E1 -8022.316,E2 -8022.316} C_VEL
LIN {X 0,Y 461.746,Z 724.837,A -85,B 0,C 180,E1 -8023.197,E2 -8023.197} C_VEL
LIN {X 0,Y 462.21,Z 713.425,A -85,B 0,C 180,E1 -8023.968,E2 -8023.968} C_VEL
LIN {X 0,Y 462.663,Z 701.552,A -85,B 0,C 180,E1 -8024.571,E2 -8024.571} C_VEL
LIN {X 0,Y 463.149,Z 686.606,A -85,B 0,C 180,E1 -8025.118,E2 -8025.118} C_VEL
LIN {X 0,Y 463.455,Z 673.759,A -85,B 0,C 180,E1 -8025.417,E2 -8025.417} C_VEL
LIN {X 0,Y 464.15,Z 590.243,A -85,B 0,C 180,E1 -8026.813,E2 -8026.813} C_VEL
LIN {X 0,Y 461.444,Z 569.969,A -85,B 0,C 180,E1 -8027.285,E2 -8027.285} C_VEL
LIN {X 0,Y 462.245,Z 549.684,A -85,B 0,C 180,E1 -8030.468,E2 -8030.468} C_VEL
LIN {X 0,Y 463.05,Z 532.217,A -85,B 0,C 180,E1 -8033.242,E2 -8033.242} C_VEL
LIN {X 0,Y 463.726,Z 517.645,A -85,B 0,C 180,E1 -8035.59,E2 -8035.59} C_VEL
LIN {X 0,Y 461.121,Z 504.637,A -85,B 0,C 180,E1 -8037.873,E2 -8037.873} C_VEL
LIN {X 0,Y 460.577,Z 502.115,A -85,B 0,C 180,E1 -8038.355,E2 -8038.355} C_VEL
LIN {X 0,Y 460.52,Z 502.124,A -85,B 0,C 180,E1 -8041.282,E2 -8041.282} C_VEL
LIN {X 0,Y 460.529,Z 502.117,A -85,B 0,C 180,E1 -8044.505,E2 -8044.505} C_VEL
LIN {X 0,Y 460.498,Z 502.104,A -85,B 0,C 180,E1 -8047.622,E2 -8047.622} C_VEL
LIN {X 0,Y 460.539,Z 502.112,A -85,B 0,C 180,E1 -8050.269,E2 -8050.269} C_VEL
LIN {X 0,Y 460.509,Z 502.119,A -85,B 0,C 180,E1 -8053.373,E2 -8053.373} C_VEL
LIN {X 0,Y 460.495,Z 502.123,A -85,B 0,C 180,E1 -8056.624,E2 -8056.624} C_VEL
LIN {X 0,Y 460.551,Z 502.115,A -85,B 0,C 180,E1 -8059.728,E2 -8059.728} C_VEL
LIN {X 0,Y 460.521,Z 502.116,A -85,B 0,C 180,E1 -8062.519,E2 -8062.519} C_VEL
LIN {X 0,Y 460.542,Z 502.117,A -85,B 0,C 180,E1 -8065.623,E2 -8065.623} C_VEL
LIN {X 0,Y 460.529,Z 502.115,A -85,B 0,C 180,E1 -8068.744,E2 -8068.744} C_VEL
LIN {X 0,Y 460.551,Z 502.114,A -85,B 0,C 180,E1 -8071.767,E2 -8071.767} C_VEL
LIN {X 0,Y 460.551,Z 502.113,A -85,B 0,C 180,E1 -8074.705,E2 -8074.705} C_VEL
LIN {X 0,Y 460.503,Z 502.119,A -85,B 0,C 180,E1 -8077.571,E2 -8077.571} C_VEL
LIN {X 0,Y 460.56,Z 502.111,A -85,B 0,C 180,E1 -8080.384,E2 -8080.384} C_VEL
LIN {X 0,Y 460.556,Z 502.106,A -85,B 0,C 180,E1 -8083.146,E2 -8083.146} C_VEL
LIN {X 0,Y 460.545,Z 502.112,A -85,B 0,C 180,E1 -8085.868,E2 -8085.868} C_VEL
LIN {X 0,Y 460.623,Z 502.105,A -85,B 0,C 180,E1 -8088.56,E2 -8088.56} C_VEL
LIN {X 0,Y 460.685,Z 502.084,A -85,B 0,C 180,E1 -8092.109,E2 -8092.109} C_VEL
LIN {X 0,Y 460.697,Z 502.095,A -85,B 0,C 180,E1 -8094.748,E2 -8094.748} C_VEL
LIN {X 0,Y 460.816,Z 502.08,A -85,B 0,C 180,E1 -8097.378,E2 -8097.378} C_VEL
LIN {X 0,Y 460.844,Z 502.061,A -85,B 0,C 180,E1 -8100,E2 -8100} C_VEL
LIN {X 0,Y 460.817,Z 502.078,A -85,B 0,C 180,E1 -8102.623,E2 -8102.623} C_VEL
LIN {X 0,Y 460.709,Z 502.09,A -85,B 0,C 180,E1 -8106.13,E2 -8106.13} C_VEL
LIN {X 0,Y 460.621,Z 502.095,A -85,B 0,C 180,E1 -8108.777,E2 -8108.777} C_VEL
LIN {X 0,Y 460.604,Z 502.107,A -85,B 0,C 180,E1 -8112.445,E2 -8112.445} C_VEL
LIN {X 0,Y 460.591,Z 502.096,A -85,B 0,C 180,E1 -8115.998,E2 -8115.998} C_VEL
LIN {X 0,Y 460.563,Z 502.114,A -85,B 0,C 180,E1 -8118.903,E2 -8118.903} C_VEL
LIN {X 0,Y 460.508,Z 502.117,A -85,B 0,C 180,E1 -8121.486,E2 -8121.486} C_VEL
LIN {X 0,Y 460.535,Z 502.109,A -85,B 0,C 180,E1 -8124.333,E2 -8124.333} C_VEL
LIN {X 0,Y 460.578,Z 502.113,A -85,B 0,C 180,E1 -8127.244,E2 -8127.244} C_VEL
LIN {X 0,Y 460.525,Z 502.111,A -85,B 0,C 180,E1 -8130.239,E2 -8130.239} C_VEL
LIN {X 0,Y 460.524,Z 502.118,A -85,B 0,C 180,E1 -8133.326,E2 -8133.326} C_VEL
LIN {X 0,Y 460.476,Z 502.124,A -85,B 0,C 180,E1 -8136.53,E2 -8136.53} C_VEL
LIN {X 0,Y 460.542,Z 502.119,A -85,B 0,C 180,E1 -8138.899,E2 -8138.899} C_VEL
LIN {X 0,Y 460.519,Z 502.12,A -85,B 0,C 180,E1 -8142.182,E2 -8142.182} C_VEL
LIN {X 0,Y 460.52,Z 502.121,A -85,B 0,C 180,E1 -8145.413,E2 -8145.413} C_VEL
LIN {X 0,Y 460.534,Z 502.117,A -85,B 0,C 180,E1 -8148.398,E2 -8148.398} C_VEL
LIN {X 0,Y 460.526,Z 502.12,A -85,B 0,C 180,E1 -8151.268,E2 -8151.268} C_VEL
LIN {X 0,Y 460.51,Z 502.12,A -85,B 0,C 180,E1 -8154.555,E2 -8154.555} C_VEL
LIN {X 0,Y 460.532,Z 502.113,A -85,B 0,C 180,E1 -8157.717,E2 -8157.717} C_VEL
LIN {X 0,Y 460.542,Z 502.118,A -85,B 0,C 180,E1 -8160.77,E2 -8160.77} C_VEL
LIN {X 0,Y 460.645,Z 502.157,A -85,B 0,C 180,E1 -8162.884,E2 -8162.884} C_VEL
LIN {X 0,Y 462.618,Z 512.613,A -85,B 0,C 180,E1 -8164.827,E2 -8164.827} C_VEL
LIN {X 0,Y 462.633,Z 519.402,A -85,B 0,C 180,E1 -8166.024,E2 -8166.024} C_VEL
LIN {X 0,Y 462.041,Z 537.017,A -85,B 0,C 180,E1 -8169.057,E2 -8169.057} C_VEL
LIN {X 0,Y 461.799,Z 547.203,A -85,B 0,C 180,E1 -8170.751,E2 -8170.751} C_VEL
LIN {X 0,Y 464.607,Z 563.238,A -85,B 0,C 180,E1 -8171.126,E2 -8171.126} C_VEL
LIN {X 0,Y 464.499,Z 578.287,A -85,B 0,C 180,E1 -8171.361,E2 -8171.361} C_VEL
LIN {X 0,Y 463.719,Z 584.135,A -85,B 0,C 180,E1 -8171.425,E2 -8171.425} C_VEL
LIN {X 0,Y 458.089,Z 603.144,A -85,B 0,C 180,E1 -8171.512,E2 -8171.512} C_VEL
LIN {X 0,Y 457.503,Z 608.983,A -85,B 0,C 180,E1 -8171.584,E2 -8171.584} C_VEL
LIN {X 0,Y 456.931,Z 657.025,A -85,B 0,C 180,E1 -8172.365,E2 -8172.365} C_VEL
LIN {X 0,Y 456.657,Z 669.729,A -85,B 0,C 180,E1 -8172.74,E2 -8172.74} C_VEL
LIN {X 0,Y 456.24,Z 682.826,A -85,B 0,C 180,E1 -8173.328,E2 -8173.328} C_VEL
LIN {X 0,Y 455.743,Z 694.011,A -85,B 0,C 180,E1 -8174,E2 -8174} C_VEL
LIN {X 0,Y 455.171,Z 705.61,A -85,B 0,C 180,E1 -8174.897,E2 -8174.897} C_VEL
LIN {X 0,Y 454.542,Z 715.948,A -85,B 0,C 180,E1 -8175.906,E2 -8175.906} C_VEL
LIN {X 0,Y 454.059,Z 725.212,A -85,B 0,C 180,E1 -8177.02,E2 -8177.02} C_VEL
LIN {X 0,Y 453.692,Z 732.946,A -85,B 0,C 180,E1 -8178.156,E2 -8178.156} C_VEL
LIN {X 0,Y 453.213,Z 740.412,A -85,B 0,C 180,E1 -8179.502,E2 -8179.502} C_VEL
LIN {X 0,Y 452.877,Z 747.285,A -85,B 0,C 180,E1 -8181.073,E2 -8181.073} C_VEL
LIN {X 0,Y 452.705,Z 751.826,A -85,B 0,C 180,E1 -8182.417,E2 -8182.417} C_VEL
LIN {X 0,Y 452.606,Z 755.264,A -85,B 0,C 180,E1 -8183.76,E2 -8183.76} C_VEL
LIN {X 0,Y 452.556,Z 756.996,A -85,B 0,C 180,E1 -8184.654,E2 -8184.654} C_VEL
LIN {X 0,Y 452.469,Z 759.213,A -85,B 0,C 180,E1 -8186.438,E2 -8186.438} C_VEL
LIN {X 0,Y 452.504,Z 759.738,A -85,B 0,C 180,E1 -8187.329,E2 -8187.329} C_VEL
LIN {X 0,Y 452.431,Z 759.547,A -85,B 0,C 180,E1 -8189.11,E2 -8189.11} C_VEL
LIN {X 0,Y 452.437,Z 758.881,A -85,B 0,C 180,E1 -8190,E2 -8190} C_VEL
LIN {X 0,Y 452.439,Z 757.817,A -85,B 0,C 180,E1 -8190.89,E2 -8190.89} C_VEL
LIN {X 0,Y 452.54,Z 756.308,A -85,B 0,C 180,E1 -8191.78,E2 -8191.78} C_VEL
LIN {X 0,Y 452.696,Z 753.273,A -85,B 0,C 180,E1 -8193.115,E2 -8193.115} C_VEL
LIN {X 0,Y 452.834,Z 749.198,A -85,B 0,C 180,E1 -8194.451,E2 -8194.451} C_VEL
LIN {X 0,Y 453.06,Z 742.988,A -85,B 0,C 180,E1 -8196.01,E2 -8196.01} C_VEL
LIN {X 0,Y 453.47,Z 736.46,A -85,B 0,C 180,E1 -8197.298,E2 -8197.298} C_VEL
LIN {X 0,Y 453.894,Z 727.681,A -85,B 0,C 180,E1 -8198.683,E2 -8198.683} C_VEL
LIN {X 0,Y 454.401,Z 718.98,A -85,B 0,C 180,E1 -8199.795,E2 -8199.795} C_VEL
LIN {X 0,Y 454.957,Z 709.444,A -85,B 0,C 180,E1 -8200.795,E2 -8200.795} C_VEL
LIN {X 0,Y 455.434,Z 698.939,A -85,B 0,C 180,E1 -8201.685,E2 -8201.685} C_VEL
LIN {X 0,Y 455.892,Z 687.305,A -85,B 0,C 180,E1 -8202.464,E2 -8202.464} C_VEL
LIN {X 0,Y 456.44,Z 675.324,A -85,B 0,C 180,E1 -8203.07,E2 -8203.07} C_VEL
LIN {X 0,Y 456.732,Z 662.024,A -85,B 0,C 180,E1 -8203.543,E2 -8203.543} C_VEL
LIN {X 0,Y 456.974,Z 649.202,A -85,B 0,C 180,E1 -8203.819,E2 -8203.819} C_VEL
LIN {X 0,Y 457.643,Z 563.849,A -85,B 0,C 180,E1 -8205.164,E2 -8205.164} C_VEL
LIN {X 0,Y 454.785,Z 547.343,A -85,B 0,C 180,E1 -8205.546,E2 -8205.546} C_VEL
LIN {X 0,Y 455.266,Z 530.128,A -85,B 0,C 180,E1 -8208.449,E2 -8208.449} C_VEL
LIN {X 0,Y 455.808,Z 515.338,A -85,B 0,C 180,E1 -8211.007,E2 -8211.007} C_VEL
LIN {X 0,Y 453.517,Z 503.002,A -85,B 0,C 180,E1 -8213.336,E2 -8213.336} C_VEL
LIN {X 0,Y 453.509,Z 502.997,A -85,B 0,C 180,E1 -8216.705,E2 -8216.705} C_VEL
LIN {X 0,Y 453.474,Z 502.998,A -85,B 0,C 180,E1 -8219.784,E2 -8219.784} C_VEL
LIN {X 0,Y 453.491,Z 502.996,A -85,B 0,C 180,E1 -8223.188,E2 -8223.188} C_VEL
LIN {X 0,Y 453.453,Z 502.998,A -85,B 0,C 180,E1 -8226.298,E2 -8226.298} C_VEL
LIN {X 0,Y 453.489,Z 502.992,A -85,B 0,C 180,E1 -8229.449,E2 -8229.449} C_VEL
LIN {X 0,Y 453.49,Z 502.998,A -85,B 0,C 180,E1 -8232.99,E2 -8232.99} C_VEL
LIN {X 0,Y 453.474,Z 502.99,A -85,B 0,C 180,E1 -8235.779,E2 -8235.779} C_VEL
LIN {X 0,Y 453.491,Z 502.995,A -85,B 0,C 180,E1 -8239.39,E2 -8239.39} C_VEL
LIN {X 0,Y 453.469,Z 502.998,A -85,B 0,C 180,E1 -8242.222,E2 -8242.222} C_VEL
LIN {X 0,Y 453.485,Z 502.999,A -85,B 0,C 180,E1 -8245.221,E2 -8245.221} C_VEL
LIN {X 0,Y 453.576,Z 503.154,A -85,B 0,C 180,E1 -8246.395,E2 -8246.395} C_VEL
LIN {X 0,Y 453.721,Z 503.872,A -85,B 0,C 180,E1 -8246.565,E2 -8246.565} C_VEL
LIN {X 0,Y 456.963,Z 514.787,A -85,B 0,C 180,E1 -8246.882,E2 -8246.882} C_VEL
LIN {X 0,Y 457.707,Z 518.632,A -85,B 0,C 180,E1 -8246.978,E2 -8246.978} C_VEL
LIN {X 0,Y 456.596,Z 610.702,A -85,B 0,C 180,E1 -8248.573,E2 -8248.573} C_VEL
LIN {X 0,Y 456.309,Z 624.529,A -85,B 0,C 180,E1 -8249.002,E2 -8249.002} C_VEL
LIN {X 0,Y 456.04,Z 636.685,A -85,B 0,C 180,E1 -8249.559,E2 -8249.559} C_VEL
LIN {X 0,Y 455.513,Z 648.82,A -85,B 0,C 180,E1 -8250.304,E2 -8250.304} C_VEL
LIN {X 0,Y 454.995,Z 660.924,A -85,B 0,C 180,E1 -8251.264,E2 -8251.264} C_VEL
LIN {X 0,Y 454.51,Z 671.754,A -85,B 0,C 180,E1 -8252.362,E2 -8252.362} C_VEL
LIN {X 0,Y 454.031,Z 680.847,A -85,B 0,C 180,E1 -8253.497,E2 -8253.497} C_VEL
LIN {X 0,Y 453.619,Z 689.219,A -85,B 0,C 180,E1 -8254.782,E2 -8254.782} C_VEL
LIN {X 0,Y 453.283,Z 696.68,A -85,B 0,C 180,E1 -8256.226,E2 -8256.226} C_VEL
LIN {X 0,Y 453,Z 702.528,A -85,B 0,C 180,E1 -8257.66,E2 -8257.66} C_VEL
LIN {X 0,Y 452.835,Z 706.995,A -85,B 0,C 180,E1 -8259.086,E2 -8259.086} C_VEL
LIN {X 0,Y 452.72,Z 709.265,A -85,B 0,C 180,E1 -8260.03,E2 -8260.03} C_VEL
LIN {X 0,Y 452.59,Z 711.57,A -85,B 0,C 180,E1 -8261.3,E2 -8261.3} C_VEL
LIN {X 0,Y 452.52,Z 713.19,A -85,B 0,C 180,E1 -8262.837,E2 -8262.837} C_VEL
LIN {X 0,Y 452.537,Z 713.612,A -85,B 0,C 180,E1 -8264.333,E2 -8264.333} C_VEL
LIN {X 0,Y 452.535,Z 713.084,A -85,B 0,C 180,E1 -8265.612,E2 -8265.612} C_VEL
LIN {X 0,Y 452.607,Z 712.164,A -85,B 0,C 180,E1 -8266.531,E2 -8266.531} C_VEL
LIN {X 0,Y 452.75,Z 709.913,A -85,B 0,C 180,E1 -8267.937,E2 -8267.937} C_VEL
LIN {X 0,Y 452.896,Z 706.777,A -85,B 0,C 180,E1 -8269.268,E2 -8269.268} C_VEL
LIN {X 0,Y 453.085,Z 702.483,A -85,B 0,C 180,E1 -8270.626,E2 -8270.626} C_VEL
LIN {X 0,Y 453.367,Z 696.977,A -85,B 0,C 180,E1 -8271.98,E2 -8271.98} C_VEL
LIN {X 0,Y 453.772,Z 690.074,A -85,B 0,C 180,E1 -8273.329,E2 -8273.329} C_VEL
LIN {X 0,Y 454.189,Z 681.43,A -85,B 0,C 180,E1 -8274.673,E2 -8274.673} C_VEL
LIN {X 0,Y 454.648,Z 672.563,A -85,B 0,C 180,E1 -8275.789,E2 -8275.789} C_VEL
LIN {X 0,Y 455.103,Z 662.837,A -85,B 0,C 180,E1 -8276.791,E2 -8276.791} C_VEL
LIN {X 0,Y 455.627,Z 652.071,A -85,B 0,C 180,E1 -8277.679,E2 -8277.679} C_VEL
LIN {X 0,Y 456.127,Z 640.048,A -85,B 0,C 180,E1 -8278.455,E2 -8278.455} C_VEL
LIN {X 0,Y 456.465,Z 627.643,A -85,B 0,C 180,E1 -8279.062,E2 -8279.062} C_VEL
LIN {X 0,Y 456.763,Z 615.264,A -85,B 0,C 180,E1 -8279.482,E2 -8279.482} C_VEL
LIN {X 0,Y 456.92,Z 598.43,A -85,B 0,C 180,E1 -8279.825,E2 -8279.825} C_VEL
LIN {X 0,Y 458.059,Z 518.69,A -85,B 0,C 180,E1 -8281.236,E2 -8281.236} C_VEL
LIN {X 0,Y 455.943,Z 510.99,A -85,B 0,C 180,E1 -8281.478,E2 -8281.478} C_VEL
LIN {X 0,Y 454.315,Z 506.55,A -85,B 0,C 180,E1 -8281.662,E2 -8281.662} C_VEL
LIN {X 0,Y 453.758,Z 502.965,A -85,B 0,C 180,E1 -8282.663,E2 -8282.663} C_VEL
LIN {X 0,Y 453.675,Z 502.973,A -85,B 0,C 180,E1 -8286.225,E2 -8286.225} C_VEL
LIN {X 0,Y 453.584,Z 502.987,A -85,B 0,C 180,E1 -8288.913,E2 -8288.913} C_VEL
LIN {X 0,Y 453.592,Z 502.982,A -85,B 0,C 180,E1 -8292.551,E2 -8292.551} C_VEL
LIN {X 0,Y 453.535,Z 502.989,A -85,B 0,C 180,E1 -8296.196,E2 -8296.196} C_VEL
LIN {X 0,Y 453.512,Z 502.996,A -85,B 0,C 180,E1 -8299.041,E2 -8299.041} C_VEL
LIN {X 0,Y 453.468,Z 502.997,A -85,B 0,C 180,E1 -8301.836,E2 -8301.836} C_VEL
LIN {X 0,Y 453.506,Z 502.994,A -85,B 0,C 180,E1 -8304.735,E2 -8304.735} C_VEL
LIN {X 0,Y 453.531,Z 502.986,A -85,B 0,C 180,E1 -8307.962,E2 -8307.962} C_VEL
LIN {X 0,Y 453.476,Z 502.996,A -85,B 0,C 180,E1 -8310.76,E2 -8310.76} C_VEL
LIN {X 0,Y 453.471,Z 502.993,A -85,B 0,C 180,E1 -8313.913,E2 -8313.913} C_VEL
LIN {X 0,Y 453.465,Z 503.001,A -85,B 0,C 180,E1 -8317.189,E2 -8317.189} C_VEL
LIN {X 0,Y 453.501,Z 502.994,A -85,B 0,C 180,E1 -8319.449,E2 -8319.449} C_VEL
LIN {X 0,Y 453.459,Z 503.004,A -85,B 0,C 180,E1 -8322.996,E2 -8322.996} C_VEL
LIN {X 0,Y 453.469,Z 502.997,A -85,B 0,C 180,E1 -8325.781,E2 -8325.781} C_VEL
LIN {X 0,Y 453.478,Z 502.998,A -85,B 0,C 180,E1 -8328.21,E2 -8328.21} C_VEL
LIN {X 0,Y 453.507,Z 502.997,A -85,B 0,C 180,E1 -8330.792,E2 -8330.792} C_VEL
LIN {X 0,Y 453.454,Z 502.999,A -85,B 0,C 180,E1 -8333.918,E2 -8333.918} C_VEL
LIN {X 0,Y 453.481,Z 503.004,A -85,B 0,C 180,E1 -8337.152,E2 -8337.152} C_VEL
LIN {X 0,Y 453.474,Z 503.001,A -85,B 0,C 180,E1 -8340.269,E2 -8340.269} C_VEL
LIN {X 0,Y 453.536,Z 503.098,A -85,B 0,C 180,E1 -8341.534,E2 -8341.534} C_VEL
LIN {X 0,Y 455.865,Z 514.133,A -85,B 0,C 180,E1 -8343.616,E2 -8343.616} C_VEL
LIN {X 0,Y 456.596,Z 518.864,A -85,B 0,C 180,E1 -8344.471,E2 -8344.471} C_VEL
LIN {X 0,Y 455.623,Z 538.679,A -85,B 0,C 180,E1 -8347.745,E2 -8347.745} C_VEL
LIN {X 0,Y 454.692,Z 559.226,A -85,B 0,C 180,E1 -8351.06,E2 -8351.06} C_VEL
LIN {X 0,Y 454.381,Z 567.551,A -85,B 0,C 180,E1 -8352.363,E2 -8352.363} C_VEL
LIN {X 0,Y 457.496,Z 593.299,A -85,B 0,C 180,E1 -8352.97,E2 -8352.97} C_VEL
LIN {X 0,Y 456.465,Z 678.863,A -85,B 0,C 180,E1 -8354.484,E2 -8354.484} C_VEL
LIN {X 0,Y 455.922,Z 695.645,A -85,B 0,C 180,E1 -8355.009,E2 -8355.009} C_VEL
LIN {X 0,Y 455.517,Z 707.567,A -85,B 0,C 180,E1 -8355.538,E2 -8355.538} C_VEL
LIN {X 0,Y 454.967,Z 719.591,A -85,B 0,C 180,E1 -8356.261,E2 -8356.261} C_VEL
LIN {X 0,Y 454.598,Z 730.213,A -85,B 0,C 180,E1 -8357.088,E2 -8357.088} C_VEL
LIN {X 0,Y 454.045,Z 740.236,A -85,B 0,C 180,E1 -8358.052,E2 -8358.052} C_VEL
LIN {X 0,Y 453.586,Z 748.806,A -85,B 0,C 180,E1 -8359.059,E2 -8359.059} C_VEL
LIN {X 0,Y 453.257,Z 756.689,A -85,B 0,C 180,E1 -8360.18,E2 -8360.18} C_VEL
LIN {X 0,Y 452.942,Z 764.343,A -85,B 0,C 180,E1 -8361.524,E2 -8361.524} C_VEL
LIN {X 0,Y 452.718,Z 770.472,A -85,B 0,C 180,E1 -8362.866,E2 -8362.866} C_VEL
LIN {X 0,Y 452.633,Z 775.314,A -85,B 0,C 180,E1 -8364.208,E2 -8364.208} C_VEL
LIN {X 0,Y 452.531,Z 779.011,A -85,B 0,C 180,E1 -8365.546,E2 -8365.546} C_VEL
LIN {X 0,Y 452.507,Z 780.914,A -85,B 0,C 180,E1 -8366.438,E2 -8366.438} C_VEL
LIN {X 0,Y 452.578,Z 782.357,A -85,B 0,C 180,E1 -8367.33,E2 -8367.33} C_VEL
LIN {X 0,Y 452.438,Z 783.987,A -85,B 0,C 180,E1 -8369.11,E2 -8369.11} C_VEL
LIN {X 0,Y 452.449,Z 784.214,A -85,B 0,C 180,E1 -8370,E2 -8370} C_VEL
LIN {X 0,Y 452.491,Z 783.383,A -85,B 0,C 180,E1 -8371.78,E2 -8371.78} C_VEL
LIN {X 0,Y 452.579,Z 782.379,A -85,B 0,C 180,E1 -8372.67,E2 -8372.67} C_VEL
LIN {X 0,Y 452.514,Z 780.951,A -85,B 0,C 180,E1 -8373.562,E2 -8373.562} C_VEL
LIN {X 0,Y 452.568,Z 777.977,A -85,B 0,C 180,E1 -8374.899,E2 -8374.899} C_VEL
LIN {X 0,Y 452.65,Z 773.211,A -85,B 0,C 180,E1 -8376.441,E2 -8376.441} C_VEL
LIN {X 0,Y 452.853,Z 766.685,A -85,B 0,C 180,E1 -8378.029,E2 -8378.029} C_VEL
LIN {X 0,Y 453.153,Z 759.598,A -85,B 0,C 180,E1 -8379.372,E2 -8379.372} C_VEL
LIN {X 0,Y 453.516,Z 750.745,A -85,B 0,C 180,E1 -8380.717,E2 -8380.717} C_VEL
LIN {X 0,Y 454.015,Z 741.643,A -85,B 0,C 180,E1 -8381.835,E2 -8381.835} C_VEL
LIN {X 0,Y 454.456,Z 732.624,A -85,B 0,C 180,E1 -8382.744,E2 -8382.744} C_VEL
LIN {X 0,Y 454.97,Z 721.794,A -85,B 0,C 180,E1 -8383.625,E2 -8383.625} C_VEL
LIN {X 0,Y 455.501,Z 709.47,A -85,B 0,C 180,E1 -8384.406,E2 -8384.406} C_VEL
LIN {X 0,Y 455.908,Z 697.715,A -85,B 0,C 180,E1 -8384.963,E2 -8384.963} C_VEL
LIN {X 0,Y 456.332,Z 684.87,A -85,B 0,C 180,E1 -8385.378,E2 -8385.378} C_VEL
LIN {X 0,Y 456.614,Z 668.713,A -85,B 0,C 180,E1 -8385.711,E2 -8385.711} C_VEL
LIN {X 0,Y 457.293,Z 590.726,A -85,B 0,C 180,E1 -8387.044,E2 -8387.044} C_VEL
LIN {X 0,Y 454.463,Z 569.554,A -85,B 0,C 180,E1 -8387.538,E2 -8387.538} C_VEL
LIN {X 0,Y 455.264,Z 550.604,A -85,B 0,C 180,E1 -8390.56,E2 -8390.56} C_VEL
LIN {X 0,Y 456.205,Z 531.696,A -85,B 0,C 180,E1 -8393.611,E2 -8393.611} C_VEL
LIN {X 0,Y 456.827,Z 520.009,A -85,B 0,C 180,E1 -8395.515,E2 -8395.515} C_VEL
LIN {X 0,Y 455.569,Z 512.568,A -85,B 0,C 180,E1 -8396.822,E2 -8396.822} C_VEL
LIN {X 0,Y 453.528,Z 502.994,A -85,B 0,C 180,E1 -8398.572,E2 -8398.572} C_VEL
LIN {X 0,Y 453.463,Z 502.999,A -85,B 0,C 180,E1 -8401.799,E2 -8401.799} C_VEL
LIN {X 0,Y 453.477,Z 503,A -85,B 0,C 180,E1 -8404.989,E2 -8404.989} C_VEL
LIN {X 0,Y 453.461,Z 502.977,A -85,B 0,C 180,E1 -8408.311,E2 -8408.311} C_VEL
LIN {X 0,Y 453.491,Z 502.991,A -85,B 0,C 180,E1 -8410.608,E2 -8410.608} C_VEL
LIN {X 0,Y 453.472,Z 502.992,A -85,B 0,C 180,E1 -8414.219,E2 -8414.219} C_VEL
LIN {X 0,Y 453.459,Z 503.003,A -85,B 0,C 180,E1 -8417.004,E2 -8417.004} C_VEL
LIN {X 0,Y 453.524,Z 502.99,A -85,B 0,C 180,E1 -8420.554,E2 -8420.554} C_VEL
LIN {X 0,Y 453.45,Z 502.993,A -85,B 0,C 180,E1 -8423.917,E2 -8423.917} C_VEL
LIN {X 0,Y 453.476,Z 502.999,A -85,B 0,C 180,E1 -8427.151,E2 -8427.151} C_VEL
LIN {X 0,Y 453.507,Z 502.984,A -85,B 0,C 180,E1 -8430.271,E2 -8430.271} C_VEL
LIN {X 0,Y 453.506,Z 502.994,A -85,B 0,C 180,E1 -8433.294,E2 -8433.294} C_VEL
LIN {X 0,Y 453.495,Z 502.98,A -85,B 0,C 180,E1 -8436.238,E2 -8436.238} C_VEL
LIN {X 0,Y 453.475,Z 503,A -85,B 0,C 180,E1 -8439.117,E2 -8439.117} C_VEL
LIN {X 0,Y 453.502,Z 502.985,A -85,B 0,C 180,E1 -8441.944,E2 -8441.944} C_VEL
LIN {X 0,Y 453.53,Z 502.98,A -85,B 0,C 180,E1 -8444.726,E2 -8444.726} C_VEL
LIN {X 0,Y 453.593,Z 502.983,A -85,B 0,C 180,E1 -8447.472,E2 -8447.472} C_VEL
LIN {X 0,Y 453.584,Z 502.973,A -85,B 0,C 180,E1 -8451.087,E2 -8451.087} C_VEL
LIN {X 0,Y 453.675,Z 502.968,A -85,B 0,C 180,E1 -8453.775,E2 -8453.775} C_VEL
LIN {X 0,Y 453.757,Z 502.96,A -85,B 0,C 180,E1 -8457.337,E2 -8457.337} C_VEL
LIN {X 0,Y 453.814,Z 502.936,A -85,B 0,C 180,E1 -8460,E2 -8460} C_VEL
LIN {X 0,Y 453.758,Z 502.957,A -85,B 0,C 180,E1 -8462.663,E2 -8462.663} C_VEL
LIN {X 0,Y 453.676,Z 502.967,A -85,B 0,C 180,E1 -8466.226,E2 -8466.226} C_VEL
LIN {X 0,Y 453.584,Z 502.972,A -85,B 0,C 180,E1 -8468.914,E2 -8468.914} C_VEL
LIN {X 0,Y 453.554,Z 502.986,A -85,B 0,C 180,E1 -8472.529,E2 -8472.529} C_VEL
LIN {X 0,Y 453.536,Z 502.974,A -85,B 0,C 180,E1 -8476.197,E2 -8476.197} C_VEL
LIN {X 0,Y 453.513,Z 502.994,A -85,B 0,C 180,E1 -8479.042,E2 -8479.042} C_VEL
LIN {X 0,Y 453.469,Z 502.991,A -85,B 0,C 180,E1 -8481.837,E2 -8481.837} C_VEL
LIN {X 0,Y 453.507,Z 502.988,A -85,B 0,C 180,E1 -8484.735,E2 -8484.735} C_VEL
LIN {X 0,Y 453.532,Z 502.985,A -85,B 0,C 180,E1 -8487.962,E2 -8487.962} C_VEL
LIN {X 0,Y 453.479,Z 502.992,A -85,B 0,C 180,E1 -8490.76,E2 -8490.76} C_VEL
LIN {X 0,Y 453.473,Z 502.992,A -85,B 0,C 180,E1 -8493.914,E2 -8493.914} C_VEL
LIN {X 0,Y 453.467,Z 503.003,A -85,B 0,C 180,E1 -8497.189,E2 -8497.189} C_VEL
LIN {X 0,Y 453.501,Z 502.992,A -85,B 0,C 180,E1 -8499.449,E2 -8499.449} C_VEL
LIN {X 0,Y 453.466,Z 503.001,A -85,B 0,C 180,E1 -8502.995,E2 -8502.995} C_VEL
LIN {X 0,Y 453.474,Z 502.996,A -85,B 0,C 180,E1 -8505.781,E2 -8505.781} C_VEL
LIN {X 0,Y 453.493,Z 502.995,A -85,B 0,C 180,E1 -8509.392,E2 -8509.392} C_VEL
LIN {X 0,Y 453.449,Z 502.997,A -85,B 0,C 180,E1 -8512.228,E2 -8512.228} C_VEL
LIN {X 0,Y 453.487,Z 502.993,A -85,B 0,C 180,E1 -8515.224,E2 -8515.224} C_VEL
LIN {X 0,Y 453.467,Z 502.994,A -85,B 0,C 180,E1 -8518.476,E2 -8518.476} C_VEL
LIN {X 0,Y 453.534,Z 502.99,A -85,B 0,C 180,E1 -8522.041,E2 -8522.041} C_VEL
LIN {X 0,Y 453.607,Z 503.124,A -85,B 0,C 180,E1 -8522.678,E2 -8522.678} C_VEL
LIN {X 0,Y 455.652,Z 513.657,A -85,B 0,C 180,E1 -8524.659,E2 -8524.659} C_VEL
LIN {X 0,Y 455.819,Z 518.865,A -85,B 0,C 180,E1 -8525.596,E2 -8525.596} C_VEL
LIN {X 0,Y 455.111,Z 538.257,A -85,B 0,C 180,E1 -8528.96,E2 -8528.96} C_VEL
LIN {X 0,Y 454.894,Z 547.289,A -85,B 0,C 180,E1 -8530.466,E2 -8530.466} C_VEL
LIN {X 0,Y 457.865,Z 564.736,A -85,B 0,C 180,E1 -8530.883,E2 -8530.883} C_VEL
LIN {X 0,Y 457.503,Z 608.983,A -85,B 0,C 180,E1 -8531.584,E2 -8531.584} C_VEL
LIN {X 0,Y 456.891,Z 614.825,A -85,B 0,C 180,E1 -8531.655,E2 -8531.655} C_VEL
LIN {X 0,Y 451.109,Z 633.807,A -85,B 0,C 180,E1 -8531.74,E2 -8531.74} C_VEL
LIN {X 0,Y 450.374,Z 639.656,A -85,B 0,C 180,E1 -8531.807,E2 -8531.807} C_VEL
LIN {X 0,Y 450.081,Z 659.36,A -85,B 0,C 180,E1 -8532.163,E2 -8532.163} C_VEL
LIN {X 0,Y 449.792,Z 672.541,A -85,B 0,C 180,E1 -8532.601,E2 -8532.601} C_VEL
LIN {X 0,Y 449.32,Z 684.712,A -85,B 0,C 180,E1 -8533.18,E2 -8533.18} C_VEL
LIN {X 0,Y 448.82,Z 695.531,A -85,B 0,C 180,E1 -8533.863,E2 -8533.863} C_VEL
LIN {X 0,Y 448.221,Z 706.794,A -85,B 0,C 180,E1 -8534.774,E2 -8534.774} C_VEL
LIN {X 0,Y 447.557,Z 716.966,A -85,B 0,C 180,E1 -8535.797,E2 -8535.797} C_VEL
LIN {X 0,Y 447.076,Z 725.652,A -85,B 0,C 180,E1 -8536.871,E2 -8536.871} C_VEL
LIN {X 0,Y 446.636,Z 734.344,A -85,B 0,C 180,E1 -8538.197,E2 -8538.197} C_VEL
LIN {X 0,Y 446.125,Z 741.583,A -85,B 0,C 180,E1 -8539.563,E2 -8539.563} C_VEL
LIN {X 0,Y 445.843,Z 747.386,A -85,B 0,C 180,E1 -8540.931,E2 -8540.931} C_VEL
LIN {X 0,Y 445.654,Z 751.946,A -85,B 0,C 180,E1 -8542.297,E2 -8542.297} C_VEL
LIN {X 0,Y 445.532,Z 755.403,A -85,B 0,C 180,E1 -8543.661,E2 -8543.661} C_VEL
LIN {X 0,Y 445.474,Z 757.151,A -85,B 0,C 180,E1 -8544.568,E2 -8544.568} C_VEL
LIN {X 0,Y 445.369,Z 759.385,A -85,B 0,C 180,E1 -8546.381,E2 -8546.381} C_VEL
LIN {X 0,Y 445.429,Z 759.921,A -85,B 0,C 180,E1 -8547.287,E2 -8547.287} C_VEL
LIN {X 0,Y 445.342,Z 759.75,A -85,B 0,C 180,E1 -8549.096,E2 -8549.096} C_VEL
LIN {X 0,Y 445.345,Z 759.091,A -85,B 0,C 180,E1 -8550,E2 -8550} C_VEL
LIN {X 0,Y 445.35,Z 758.041,A -85,B 0,C 180,E1 -8550.904,E2 -8550.904} C_VEL
LIN {X 0,Y 445.455,Z 756.542,A -85,B 0,C 180,E1 -8551.808,E2 -8551.808} C_VEL
LIN {X 0,Y 445.621,Z 753.523,A -85,B 0,C 180,E1 -8553.164,E2 -8553.164} C_VEL
LIN {X 0,Y 445.756,Z 749.465,A -85,B 0,C 180,E1 -8554.521,E2 -8554.521} C_VEL
LIN {X 0,Y 446.028,Z 743.272,A -85,B 0,C 180,E1 -8556.105,E2 -8556.105} C_VEL
LIN {X 0,Y 446.424,Z 737.177,A -85,B 0,C 180,E1 -8557.337,E2 -8557.337} C_VEL
LIN {X 0,Y 446.788,Z 729.593,A -85,B 0,C 180,E1 -8558.594,E2 -8558.594} C_VEL
LIN {X 0,Y 447.291,Z 721.227,A -85,B 0,C 180,E1 -8559.724,E2 -8559.724} C_VEL
LIN {X 0,Y 447.946,Z 710.971,A -85,B 0,C 180,E1 -8560.852,E2 -8560.852} C_VEL
LIN {X 0,Y 448.431,Z 700.847,A -85,B 0,C 180,E1 -8561.756,E2 -8561.756} C_VEL
LIN {X 0,Y 448.966,Z 689.697,A -85,B 0,C 180,E1 -8562.544,E2 -8562.544} C_VEL
LIN {X 0,Y 449.548,Z 677.141,A -85,B 0,C 180,E1 -8563.217,E2 -8563.217} C_VEL
LIN {X 0,Y 449.847,Z 664.825,A -85,B 0,C 180,E1 -8563.697,E2 -8563.697} C_VEL
LIN {X 0,Y 450.068,Z 652.221,A -85,B 0,C 180,E1 -8564.007,E2 -8564.007} C_VEL
LIN {X 0,Y 450.822,Z 564.587,A -85,B 0,C 180,E1 -8565.41,E2 -8565.41} C_VEL
LIN {X 0,Y 447.869,Z 547.416,A -85,B 0,C 180,E1 -8565.822,E2 -8565.822} C_VEL
LIN {X 0,Y 448.342,Z 530.202,A -85,B 0,C 180,E1 -8568.744,E2 -8568.744} C_VEL
LIN {X 0,Y 448.871,Z 516.659,A -85,B 0,C 180,E1 -8571.107,E2 -8571.107} C_VEL
LIN {X 0,Y 446.488,Z 503.878,A -85,B 0,C 180,E1 -8573.541,E2 -8573.541} C_VEL
LIN {X 0,Y 446.477,Z 503.872,A -85,B 0,C 180,E1 -8577.16,E2 -8577.16} C_VEL
LIN {X 0,Y 446.429,Z 503.876,A -85,B 0,C 180,E1 -8580.249,E2 -8580.249} C_VEL
LIN {X 0,Y 446.446,Z 503.871,A -85,B 0,C 180,E1 -8583.453,E2 -8583.453} C_VEL
LIN {X 0,Y 446.401,Z 503.878,A -85,B 0,C 180,E1 -8586.744,E2 -8586.744} C_VEL
LIN {X 0,Y 446.442,Z 503.868,A -85,B 0,C 180,E1 -8590.197,E2 -8590.197} C_VEL
LIN {X 0,Y 446.445,Z 503.87,A -85,B 0,C 180,E1 -8593.602,E2 -8593.602} C_VEL
LIN {X 0,Y 446.421,Z 503.87,A -85,B 0,C 180,E1 -8596.399,E2 -8596.399} C_VEL
LIN {X 0,Y 446.444,Z 503.871,A -85,B 0,C 180,E1 -8599.802,E2 -8599.802} C_VEL
LIN {X 0,Y 446.424,Z 503.875,A -85,B 0,C 180,E1 -8602.122,E2 -8602.122} C_VEL
LIN {X 0,Y 446.439,Z 503.875,A -85,B 0,C 180,E1 -8605.477,E2 -8605.477} C_VEL
LIN {X 0,Y 446.529,Z 503.988,A -85,B 0,C 180,E1 -8606.23,E2 -8606.23} C_VEL
LIN {X 0,Y 446.576,Z 504.264,A -85,B 0,C 180,E1 -8606.295,E2 -8606.295} C_VEL
LIN {X 0,Y 450.228,Z 516.109,A -85,B 0,C 180,E1 -8606.652,E2 -8606.652} C_VEL
LIN {X 0,Y 450.878,Z 519.881,A -85,B 0,C 180,E1 -8606.746,E2 -8606.746} C_VEL
LIN {X 0,Y 449.715,Z 611.819,A -85,B 0,C 180,E1 -8608.381,E2 -8608.381} C_VEL
LIN {X 0,Y 449.423,Z 625.004,A -85,B 0,C 180,E1 -8608.801,E2 -8608.801} C_VEL
LIN {X 0,Y 449.095,Z 637.661,A -85,B 0,C 180,E1 -8609.394,E2 -8609.394} C_VEL
LIN {X 0,Y 448.566,Z 649.931,A -85,B 0,C 180,E1 -8610.168,E2 -8610.168} C_VEL
LIN {X 0,Y 448.063,Z 661.26,A -85,B 0,C 180,E1 -8611.084,E2 -8611.084} C_VEL
LIN {X 0,Y 447.57,Z 671.723,A -85,B 0,C 180,E1 -8612.15,E2 -8612.15} C_VEL
LIN {X 0,Y 447.047,Z 681.113,A -85,B 0,C 180,E1 -8613.33,E2 -8613.33} C_VEL
LIN {X 0,Y 446.614,Z 689.386,A -85,B 0,C 180,E1 -8614.607,E2 -8614.607} C_VEL
LIN {X 0,Y 446.298,Z 696.459,A -85,B 0,C 180,E1 -8615.968,E2 -8615.968} C_VEL
LIN {X 0,Y 445.996,Z 701.977,A -85,B 0,C 180,E1 -8617.289,E2 -8617.289} C_VEL
LIN {X 0,Y 445.794,Z 706.703,A -85,B 0,C 180,E1 -8618.74,E2 -8618.74} C_VEL
LIN {X 0,Y 445.691,Z 709.17,A -85,B 0,C 180,E1 -8619.701,E2 -8619.701} C_VEL
LIN {X 0,Y 445.521,Z 711.95,A -85,B 0,C 180,E1 -8621.167,E2 -8621.167} C_VEL
LIN {X 0,Y 445.451,Z 713.546,A -85,B 0,C 180,E1 -8622.556,E2 -8622.556} C_VEL
LIN {X 0,Y 445.47,Z 714.18,A -85,B 0,C 180,E1 -8624.228,E2 -8624.228} C_VEL
LIN {X 0,Y 445.47,Z 713.826,A -85,B 0,C 180,E1 -8625.379,E2 -8625.379} C_VEL
LIN {X 0,Y 445.527,Z 713.049,A -85,B 0,C 180,E1 -8626.313,E2 -8626.313} C_VEL
LIN {X 0,Y 445.673,Z 710.746,A -85,B 0,C 180,E1 -8627.871,E2 -8627.871} C_VEL
LIN {X 0,Y 445.875,Z 706.813,A -85,B 0,C 180,E1 -8629.556,E2 -8629.556} C_VEL
LIN {X 0,Y 446.099,Z 702.355,A -85,B 0,C 180,E1 -8630.935,E2 -8630.935} C_VEL
LIN {X 0,Y 446.472,Z 696.426,A -85,B 0,C 180,E1 -8632.356,E2 -8632.356} C_VEL
LIN {X 0,Y 446.853,Z 689.473,A -85,B 0,C 180,E1 -8633.679,E2 -8633.679} C_VEL
LIN {X 0,Y 447.289,Z 680.584,A -85,B 0,C 180,E1 -8635.042,E2 -8635.042} C_VEL
LIN {X 0,Y 447.799,Z 671.427,A -85,B 0,C 180,E1 -8636.175,E2 -8636.175} C_VEL
LIN {X 0,Y 448.295,Z 661.263,A -85,B 0,C 180,E1 -8637.192,E2 -8637.192} C_VEL
LIN {X 0,Y 448.868,Z 649.985,A -85,B 0,C 180,E1 -8638.093,E2 -8638.093} C_VEL
LIN {X 0,Y 449.4,Z 638.237,A -85,B 0,C 180,E1 -8638.824,E2 -8638.824} C_VEL
LIN {X 0,Y 449.741,Z 624.903,A -85,B 0,C 180,E1 -8639.434,E2 -8639.434} C_VEL
LIN {X 0,Y 450,Z 612.772,A -85,B 0,C 180,E1 -8639.813,E2 -8639.813} C_VEL
LIN {X 0,Y 451.276,Z 519.535,A -85,B 0,C 180,E1 -8641.526,E2 -8641.526} C_VEL
LIN {X 0,Y 449.57,Z 513.458,A -85,B 0,C 180,E1 -8641.725,E2 -8641.725} C_VEL
LIN {X 0,Y 447.295,Z 507.325,A -85,B 0,C 180,E1 -8641.969,E2 -8641.969} C_VEL
LIN {X 0,Y 446.612,Z 503.857,A -85,B 0,C 180,E1 -8642.988,E2 -8642.988} C_VEL
LIN {X 0,Y 446.643,Z 503.849,A -85,B 0,C 180,E1 -8646.324,E2 -8646.324} C_VEL
LIN {X 0,Y 446.53,Z 503.866,A -85,B 0,C 180,E1 -8649.055,E2 -8649.055} C_VEL
LIN {X 0,Y 446.525,Z 503.863,A -85,B 0,C 180,E1 -8652.729,E2 -8652.729} C_VEL
LIN {X 0,Y 446.481,Z 503.868,A -85,B 0,C 180,E1 -8656.459,E2 -8656.459} C_VEL
LIN {X 0,Y 446.461,Z 503.874,A -85,B 0,C 180,E1 -8659.303,E2 -8659.303} C_VEL
LIN {X 0,Y 446.41,Z 503.875,A -85,B 0,C 180,E1 -8662.2,E2 -8662.2} C_VEL
LIN {X 0,Y 446.45,Z 503.874,A -85,B 0,C 180,E1 -8665.153,E2 -8665.153} C_VEL
LIN {X 0,Y 446.477,Z 503.864,A -85,B 0,C 180,E1 -8668.179,E2 -8668.179} C_VEL
LIN {X 0,Y 446.413,Z 503.875,A -85,B 0,C 180,E1 -8671.301,E2 -8671.301} C_VEL
LIN {X 0,Y 446.424,Z 503.872,A -85,B 0,C 180,E1 -8674.523,E2 -8674.523} C_VEL
LIN {X 0,Y 446.427,Z 503.872,A -85,B 0,C 180,E1 -8678.083,E2 -8678.083} C_VEL
LIN {X 0,Y 446.422,Z 503.879,A -85,B 0,C 180,E1 -8680.918,E2 -8680.918} C_VEL
LIN {X 0,Y 446.397,Z 503.877,A -85,B 0,C 180,E1 -8683.847,E2 -8683.847} C_VEL
LIN {X 0,Y 446.417,Z 503.877,A -85,B 0,C 180,E1 -8686.401,E2 -8686.401} C_VEL
LIN {X 0,Y 446.444,Z 503.874,A -85,B 0,C 180,E1 -8689.803,E2 -8689.803} C_VEL
LIN {X 0,Y 446.425,Z 503.875,A -85,B 0,C 180,E1 -8692.124,E2 -8692.124} C_VEL
LIN {X 0,Y 446.428,Z 503.878,A -85,B 0,C 180,E1 -8695.478,E2 -8695.478} C_VEL
LIN {X 0,Y 446.415,Z 503.884,A -85,B 0,C 180,E1 -8698.7,E2 -8698.7} C_VEL
LIN {X 0,Y 446.504,Z 503.914,A -85,B 0,C 180,E1 -8701.215,E2 -8701.215} C_VEL
LIN {X 0,Y 449.098,Z 516.243,A -85,B 0,C 180,E1 -8703.601,E2 -8703.601} C_VEL
LIN {X 0,Y 449.731,Z 521.473,A -85,B 0,C 180,E1 -8704.549,E2 -8704.549} C_VEL
LIN {X 0,Y 448.595,Z 541.495,A -85,B 0,C 180,E1 -8707.914,E2 -8707.914} C_VEL
LIN {X 0,Y 447.623,Z 561.658,A -85,B 0,C 180,E1 -8711.225,E2 -8711.225} C_VEL
LIN {X 0,Y 447.377,Z 566.648,A -85,B 0,C 180,E1 -8712.031,E2 -8712.031} C_VEL
LIN {X 0,Y 450.727,Z 592.392,A -85,B 0,C 180,E1 -8712.676,E2 -8712.676} C_VEL
LIN {X 0,Y 449.656,Z 677.278,A -85,B 0,C 180,E1 -8714.214,E2 -8714.214} C_VEL
LIN {X 0,Y 449.066,Z 695.251,A -85,B 0,C 180,E1 -8714.774,E2 -8714.774} C_VEL
LIN {X 0,Y 448.628,Z 707.222,A -85,B 0,C 180,E1 -8715.311,E2 -8715.311} C_VEL
LIN {X 0,Y 448.063,Z 719.292,A -85,B 0,C 180,E1 -8716.045,E2 -8716.045} C_VEL
LIN {X 0,Y 447.605,Z 730.737,A -85,B 0,C 180,E1 -8716.955,E2 -8716.955} C_VEL
LIN {X 0,Y 447.017,Z 741.033,A -85,B 0,C 180,E1 -8717.977,E2 -8717.977} C_VEL
LIN {X 0,Y 446.485,Z 750.244,A -85,B 0,C 180,E1 -8719.112,E2 -8719.112} C_VEL
LIN {X 0,Y 446.069,Z 759.182,A -85,B 0,C 180,E1 -8720.478,E2 -8720.478} C_VEL
LIN {X 0,Y 445.782,Z 766.339,A -85,B 0,C 180,E1 -8721.843,E2 -8721.843} C_VEL
LIN {X 0,Y 445.602,Z 772.177,A -85,B 0,C 180,E1 -8723.252,E2 -8723.252} C_VEL
LIN {X 0,Y 445.533,Z 776.464,A -85,B 0,C 180,E1 -8724.569,E2 -8724.569} C_VEL
LIN {X 0,Y 445.453,Z 778.802,A -85,B 0,C 180,E1 -8725.476,E2 -8725.476} C_VEL
LIN {X 0,Y 445.407,Z 780.707,A -85,B 0,C 180,E1 -8726.381,E2 -8726.381} C_VEL
LIN {X 0,Y 445.497,Z 782.157,A -85,B 0,C 180,E1 -8727.287,E2 -8727.287} C_VEL
LIN {X 0,Y 445.349,Z 783.792,A -85,B 0,C 180,E1 -8729.096,E2 -8729.096} C_VEL
LIN {X 0,Y 445.356,Z 784.022,A -85,B 0,C 180,E1 -8730,E2 -8730} C_VEL
LIN {X 0,Y 445.408,Z 783.2,A -85,B 0,C 180,E1 -8731.808,E2 -8731.808} C_VEL
LIN {X 0,Y 445.498,Z 782.198,A -85,B 0,C 180,E1 -8732.713,E2 -8732.713} C_VEL
LIN {X 0,Y 445.412,Z 780.776,A -85,B 0,C 180,E1 -8733.619,E2 -8733.619} C_VEL
LIN {X 0,Y 445.5,Z 777.808,A -85,B 0,C 180,E1 -8734.977,E2 -8734.977} C_VEL
LIN {X 0,Y 445.569,Z 773.451,A -85,B 0,C 180,E1 -8736.431,E2 -8736.431} C_VEL
LIN {X 0,Y 445.742,Z 767.545,A -85,B 0,C 180,E1 -8737.93,E2 -8737.93} C_VEL
LIN {X 0,Y 446.04,Z 760.746,A -85,B 0,C 180,E1 -8739.294,E2 -8739.294} C_VEL
LIN {X 0,Y 446.425,Z 752.25,A -85,B 0,C 180,E1 -8740.66,E2 -8740.66} C_VEL
LIN {X 0,Y 446.932,Z 743.488,A -85,B 0,C 180,E1 -8741.796,E2 -8741.796} C_VEL
LIN {X 0,Y 447.475,Z 733.267,A -85,B 0,C 180,E1 -8742.875,E2 -8742.875} C_VEL
LIN {X 0,Y 448.058,Z 721.752,A -85,B 0,C 180,E1 -8743.839,E2 -8743.839} C_VEL
LIN {X 0,Y 448.635,Z 709.472,A -85,B 0,C 180,E1 -8744.631,E2 -8744.631} C_VEL
LIN {X 0,Y 449.08,Z 697.799,A -85,B 0,C 180,E1 -8745.196,E2 -8745.196} C_VEL
LIN {X 0,Y 449.493,Z 685.088,A -85,B 0,C 180,E1 -8745.618,E2 -8745.618} C_VEL
LIN {X 0,Y 449.74,Z 668.829,A -85,B 0,C 180,E1 -8745.929,E2 -8745.929} C_VEL
LIN {X 0,Y 450.478,Z 591.566,A -85,B 0,C 180,E1 -8747.267,E2 -8747.267} C_VEL
LIN {X 0,Y 447.44,Z 569.11,A -85,B 0,C 180,E1 -8747.804,E2 -8747.804} C_VEL
LIN {X 0,Y 448.312,Z 550.044,A -85,B 0,C 180,E1 -8750.894,E2 -8750.894} C_VEL
LIN {X 0,Y 449.248,Z 532.569,A -85,B 0,C 180,E1 -8753.755,E2 -8753.755} C_VEL
LIN {X 0,Y 449.89,Z 520.906,A -85,B 0,C 180,E1 -8755.689,E2 -8755.689} C_VEL
LIN {X 0,Y 447.594,Z 508.955,A -85,B 0,C 180,E1 -8757.847,E2 -8757.847} C_VEL
LIN {X 0,Y 446.489,Z 503.871,A -85,B 0,C 180,E1 -8758.828,E2 -8758.828} C_VEL
LIN {X 0,Y 446.421,Z 503.876,A -85,B 0,C 180,E1 -8762.361,E2 -8762.361} C_VEL
LIN {X 0,Y 446.416,Z 503.875,A -85,B 0,C 180,E1 -8765.625,E2 -8765.625} C_VEL
LIN {X 0,Y 446.456,Z 503.855,A -85,B 0,C 180,E1 -8769.025,E2 -8769.025} C_VEL
LIN {X 0,Y 446.43,Z 503.875,A -85,B 0,C 180,E1 -8772.603,E2 -8772.603} C_VEL
LIN {X 0,Y 446.45,Z 503.874,A -85,B 0,C 180,E1 -8775.102,E2 -8775.102} C_VEL
LIN {X 0,Y 446.43,Z 503.868,A -85,B 0,C 180,E1 -8778.609,E2 -8778.609} C_VEL
LIN {X 0,Y 446.466,Z 503.873,A -85,B 0,C 180,E1 -8780.975,E2 -8780.975} C_VEL
LIN {X 0,Y 446.415,Z 503.87,A -85,B 0,C 180,E1 -8784.374,E2 -8784.374} C_VEL
LIN {X 0,Y 446.416,Z 503.872,A -85,B 0,C 180,E1 -8787.638,E2 -8787.638} C_VEL
LIN {X 0,Y 446.462,Z 503.865,A -85,B 0,C 180,E1 -8790.792,E2 -8790.792} C_VEL
LIN {X 0,Y 446.47,Z 503.865,A -85,B 0,C 180,E1 -8793.848,E2 -8793.848} C_VEL
LIN {X 0,Y 446.42,Z 503.864,A -85,B 0,C 180,E1 -8796.823,E2 -8796.823} C_VEL
LIN {X 0,Y 446.436,Z 503.872,A -85,B 0,C 180,E1 -8799.737,E2 -8799.737} C_VEL
LIN {X 0,Y 446.455,Z 503.864,A -85,B 0,C 180,E1 -8802.597,E2 -8802.597} C_VEL
LIN {X 0,Y 446.46,Z 503.871,A -85,B 0,C 180,E1 -8805.412,E2 -8805.412} C_VEL
LIN {X 0,Y 446.531,Z 503.859,A -85,B 0,C 180,E1 -8808.194,E2 -8808.194} C_VEL
LIN {X 0,Y 446.591,Z 503.839,A -85,B 0,C 180,E1 -8811.858,E2 -8811.858} C_VEL
LIN {X 0,Y 446.644,Z 503.844,A -85,B 0,C 180,E1 -8814.583,E2 -8814.583} C_VEL
